// TIA Portal V20 program export: 0 tag tables, 0 data types, 60 data blocks, 132 code blocks (in call order from the OBs), 4 instance data blocks

DATA_BLOCK "DB198_eventos_generados_routing_JDT1"   // DB198
{ S7_Optimized_Access := 'FALSE' }
// stored: AutoNumber false
   VAR
      evento : Array[0..100] of String;
   END_VAR
BEGIN
END_DATA_BLOCK

DATA_BLOCK "DB202_RegEtiquetas_1001_2000"   // DB202
{ S7_Optimized_Access := 'FALSE' }
AUTHOR : ROUTER
NAME : 20130623
VERSION : 3.1
// stored: AutoNumber false
   VAR
      Reg_Etiqueta { S7_SetPoint := 'True'} : Array[1.."ROUT_Cantidad_Etiquetas_DB"] of "ROUT_Reg_Etiqueta";
   END_VAR
BEGIN
END_DATA_BLOCK

DATA_BLOCK "DB210_DB_Eventos_Router"   // DB210
{ S7_Optimized_Access := 'FALSE' }
// stored: AutoNumber false
   VAR
      EVENTO : Array[1..2600] of Char;
   END_VAR
BEGIN
END_DATA_BLOCK

DATA_BLOCK "DB211_Lecturas_Scanner"   // DB211
{ S7_Optimized_Access := 'FALSE' }
AUTHOR : ROUTER
NAME : 20130623
VERSION : 3.1
// stored: AutoNumber false
   VAR RETAIN
      Lec_Scanner { S7_SetPoint := 'True'} : Array[0.."ROUT_Max_Scanners"] of "ROUT_Datos_Lectura_Scanner";   // Num. Escaner, Long Etiquetas leidas + 1 (Primer caracter='N' nueva etiqueta).
   END_VAR
BEGIN
END_DATA_BLOCK

DATA_BLOCK "DB212_Cola_Activa"   // DB212
{ S7_Optimized_Access := 'FALSE' }
AUTHOR : ROUTER
NAME : 20130623
VERSION : 3.1
// stored: AutoNumber false
   VAR
      Cola : Array[0..9999] of UInt;   // Valor de las diferentes colas
   END_VAR
BEGIN
END_DATA_BLOCK

DATA_BLOCK "DB213_FIFO_ORDENES_SCR"   // DB213
{ S7_Optimized_Access := 'FALSE' }
AUTHOR : ROUTER
NAME : 20130623
VERSION : 3.1
// stored: AutoNumber false
   VAR
      FIFO { S7_SetPoint := 'True'} : Array[0.."ROUT_Max_Scanners"] of "ROUT_Orden_Fifo_Scanner";   // 0 a 50 scanners y 1 ordenes posibles en la FIFO
   END_VAR
BEGIN
END_DATA_BLOCK

DATA_BLOCK "DB214_CNT_Mens_SCR"   // DB214
{ S7_Optimized_Access := 'FALSE' }
AUTHOR : ROUTER
NAME : 20130623
VERSION : 3.1
// stored: AutoNumber false
   VAR RETAIN
      RedScanners : Array[1..5] of Struct
         CNT_NODO_PROF_SCR : Array[0..254] of Byte;   // No puedo acceder directamente a cargar una dirección PA de los scanners.
      END_STRUCT;
   END_VAR
BEGIN
END_DATA_BLOCK

DATA_BLOCK "DB1_SalidasExterioresDeMesa"   // DB1
{ S7_Optimized_Access := 'FALSE' }
   VAR
      Mesa { S7_SetPoint := 'True'} : Array[0.."CTE_MaxMesas"] of "UDT_SalidasExterioresDeMesa";
   END_VAR
BEGIN
END_DATA_BLOCK

DATA_BLOCK "DB220_FIFO_ORDENES_S2"   // DB220
{ S7_Optimized_Access := 'FALSE' }
AUTHOR : ROUTER
NAME : 20130623
VERSION : 3.1
// stored: AutoNumber false
   VAR
      FIFO : Array[0.."CTE_MaxMesas"] of Struct   // 0 a 50 scanners y 1 ordenes posibles en la FIFO
         Posicion { S7_SetPoint := 'True'} : Array[1..5] of "ROUT_Orden_Fifo_Scanner";
      END_STRUCT;
   END_VAR
BEGIN
END_DATA_BLOCK

DATA_BLOCK "DB230_CONTADORES"   // DB230
{ S7_Optimized_Access := 'FALSE' }
AUTHOR : ROUTER
// stored: AutoNumber false
   VAR
      Mesa : Array[0.."CTE_MaxMesas"] of Struct
         CNT_PRESENCIA : UDInt;
         CNT_AUSENCIA_ENTRADA : UDInt;
         CNT_AUSENCIA_SALIDA : UDInt;
         CNT_PARO : UDInt;
         CNT_Seg_HB_Avance : UDInt;
         CNT_Separacion_Sal : UDInt;
         CNT_Separacion_entrada : UDInt;
         CNT_CaraDelantera : UDInt;
         CNT_Reparto_E1 : UDInt;
         CNT_Reparto_E2 : UDInt;
         CNT_Reparto_E4 : UDInt;
         CNT_Detector_Fuera : UDInt;
         AUX_CNT : UDInt;
         CNT_Bloqueo_Movimiento : UDInt;
         CNT_Reposo : UDInt;
         CNT_Atasco : UDInt;
         CNT_Gap : UDInt;
         CNT_Acumulacion : UDInt;
         TMP_En_tension : UDInt;
         CNT_TopeE1S3 : UDInt;
         CNT_TopeE2S4 : UDInt;
         CNT_Transfer : UDInt;
         TMP_Decel_SM_E1S3 : UDInt;
         TMP_Decel_SM_E2S4 : UDInt;
         TMP_Decel_SM_ELEV : UDInt;
         MEM_OCUPACION : USInt;
      END_STRUCT;
   END_VAR
BEGIN
END_DATA_BLOCK

DATA_BLOCK "DB300_VelocidadesMotores"   // DB300
{ S7_Optimized_Access := 'FALSE' }
// stored: AutoNumber false
   VAR RETAIN
      TipoMotor { S7_SetPoint := 'True'} : Array[0..50] of "VelMotor";
   END_VAR
BEGIN
END_DATA_BLOCK

DATA_BLOCK "DB702_JDT02RecepMensaje"   // DB702
{ S7_Optimized_Access := 'FALSE' }
AUTHOR : TRACKING
NAME : 20130301
VERSION : 3.0
// stored: AutoNumber false
   VAR
      Mensaje : Array[0..9999] of Char;
   END_VAR
BEGIN
END_DATA_BLOCK

DATA_BLOCK "DB703_JDT02EmisionMensaje"   // DB703
{ S7_Optimized_Access := 'FALSE' }
AUTHOR : TRACKING
NAME : 20130301
VERSION : 3.0
// stored: AutoNumber false
   VAR
      Mensaje : Array[0..9999] of Char;
   END_VAR
BEGIN
END_DATA_BLOCK

DATA_BLOCK "DB704_JDT02UltimoRecibido"   // DB704
{ S7_Optimized_Access := 'FALSE' }
AUTHOR : TRACKING
NAME : 20130301
VERSION : 3.0
// stored: AutoNumber false
   VAR
      Mensaje : Array[0..9999] of Char;
   END_VAR
BEGIN
END_DATA_BLOCK

DATA_BLOCK "DB707_JDT02EventosGenerados"   // DB707
{ S7_Optimized_Access := 'FALSE' }
AUTHOR : TRACKING
NAME : 20130301
VERSION : 3.0
// stored: AutoNumber false
   VAR
      Mensaje : Array[0..9999] of Char;
   END_VAR
BEGIN
END_DATA_BLOCK

DATA_BLOCK "DB708_JDT02EventosRecibidos"   // DB708
{ S7_Optimized_Access := 'FALSE' }
AUTHOR : TRACKING
NAME : 20130301
VERSION : 3.0
// stored: AutoNumber false
   VAR
      Mensaje : Array[0..9999] of Char;
   END_VAR
BEGIN
END_DATA_BLOCK

DATA_BLOCK "DB803_JDT01EmisionMensaje"   // DB803
{ S7_Optimized_Access := 'FALSE' }
AUTHOR : TRACKING
NAME : 20130301
VERSION : 3.0
// stored: AutoNumber false
   VAR
      Mensaje : Array[0..9999] of Char;
   END_VAR
BEGIN
END_DATA_BLOCK

DATA_BLOCK "DB804_JDT01UltimoRecibido"   // DB804
{ S7_Optimized_Access := 'FALSE' }
AUTHOR : TRACKING
NAME : 20130301
VERSION : 3.0
// stored: AutoNumber false
   VAR
      Mensaje : Array[0..9999] of Char;
   END_VAR
BEGIN
END_DATA_BLOCK

DATA_BLOCK "DB807_JDT01EventosRecibidos"   // DB807
{ S7_Optimized_Access := 'FALSE' }
AUTHOR : TRACKING
NAME : 20130301
VERSION : 3.0
// stored: AutoNumber false
   VAR
      Mensaje : Array[0..9999] of Char;
   END_VAR
BEGIN
END_DATA_BLOCK

DATA_BLOCK "DB808_JDT01EventosGenerados"   // DB808
{ S7_Optimized_Access := 'FALSE' }
AUTHOR : TRACKING
NAME : 20130301
VERSION : 3.0
// stored: AutoNumber false
   VAR
      Mensaje : Array[0..9999] of Char;
   END_VAR
BEGIN
END_DATA_BLOCK

DATA_BLOCK "DB813_UTs_Ruta"   // DB813
{ S7_Optimized_Access := 'FALSE' }
AUTHOR : TRACKING
NAME : 20130301
VERSION : 3.0
// stored: AutoNumber false
   VAR
      UT { S7_SetPoint := 'True'} : Array[0.."CTE_MaxUTs"] of "UDT_UTs_Ruta";   // Array de UT's - Ruta de la UT
   END_VAR
BEGIN
END_DATA_BLOCK

DATA_BLOCK "DB814_UTs_Etiqueta"   // DB814
{ S7_Optimized_Access := 'FALSE' }
AUTHOR : TRACKING
NAME : 20130301
VERSION : 3.0
// stored: AutoNumber false
   VAR
      UT { S7_SetPoint := 'True'} : Array[0.."CTE_MaxUTs"] of "UDT_UTs_Etiqueta";   // Array de UT's - Ruta de la UT
   END_VAR
BEGIN
END_DATA_BLOCK

DATA_BLOCK "DB816_UTs_TextoPantalla"   // DB816
{ S7_Optimized_Access := 'FALSE' }
AUTHOR : TRACKING
NAME : 20130301
VERSION : 3.0
// stored: AutoNumber false
   VAR
      UT { S7_SetPoint := 'True'} : Array[0.."CTE_MaxUTs"] of "UDT_UTs_TextoPantalla";   // Array de UT's - Ruta de la UT
   END_VAR
BEGIN
END_DATA_BLOCK

DATA_BLOCK "DB820_UTs_DatosQUBIQA"   // DB820
{ S7_Optimized_Access := 'FALSE' }
AUTHOR : TRACKING
NAME : 20130301
VERSION : 3.0
// stored: AutoNumber false
   VAR
      UT { S7_SetPoint := 'True'} : Array[0.."CTE_MaxUTs"] of "UDT_UTs_DatosQUBIQA";   // Array de UT's - Ruta de la UT
   END_VAR
BEGIN
END_DATA_BLOCK

DATA_BLOCK "DB842_EmisionPantalla"   // DB842
{ S7_Optimized_Access := 'FALSE' }
// stored: AutoNumber false
BEGIN
END_DATA_BLOCK

DATA_BLOCK "DB843_RecepcionPantalla"   // DB843
{ S7_Optimized_Access := 'FALSE' }
AUTHOR : TRACKING
NAME : 20130301
VERSION : 3.0
// stored: AutoNumber false
   VAR
      Mesa { S7_SetPoint := 'True'} : Array[0.."CTE_MaxMesas"] of "UDT_ProtocoloRecDispositivo";   // Variable provisional
   END_VAR
BEGIN
END_DATA_BLOCK

DATA_BLOCK "DB891_VariablesTCP"   // DB891
{ S7_Optimized_Access := 'FALSE' }
AUTHOR : TRACKING
NAME : 20130301
VERSION : 3.0
// stored: AutoNumber false
   VAR
      TCON_JdT_PLC_Req : Bool;
      TCON_JdT_PLC_Done : Bool;
      TCON_JdT_PLC_Busy : Bool;
      TCON_JdT_PLC_Error : Bool;
      TCON_JdT_PLC_Flanco : Bool;
      Bit_05 : Bool;
      Bit_06 : Bool;
      Bit_07 : Bool;
      TDISCON_JdT_PLC_Req : Bool;
      TDISCON_JdT_PLC_Done : Bool;
      TDISCON_JdT_PLC_Busy : Bool;
      TDISCON_JdT_PLC_Error : Bool;
      TDISCON_JdT_PLC_Flanco : Bool;
      Bit_15 : Bool;
      Bit_16 : Bool;
      Bit_17 : Bool;
      TSEND_JdT_PLC_Req : Bool := TRUE;
      TSEND_JdT_PLC_Done : Bool;
      TSEND_JdT_PLC_Busy : Bool;
      TSEND_JdT_PLC_Error : Bool;
      TSEND_JdT_PLC_Flanco : Bool;
      Bit_25 : Bool;
      Bit_26 : Bool;
      Bit_27 : Bool;
      TRCV_JdT_PLC_Req : Bool;
      TRCV_JdT_PLC_Done : Bool;
      TRCV_JdT_PLC_Busy : Bool;
      TRCV_JdT_PLC_Error : Bool;
      Bit_34 : Bool;
      Bit_35 : Bool;
      Bit_36 : Bool;
      Bit_37 : Bool;
      TCON_JdT_PLC_Status : Word;
      TDISCON_JdT_PLC_Status : Word;
      TSEND_JdT_PLC_Status : Word;
      TRCV_JdT_PLC_Status : Word;
      TCON_JdT_PLC_MStatus : Word;
      TDISCON_JdT_PLC_MStatus : Word;
      TSEND_JdT_PLC_MStatus : Word;
      TRCV_JdT_PLC_MStatus : Word;
      TSEND_JdT_PLC_Longitud : Int;
      TRCV_JdT_PLC_Longitud : Int;
      TCON_JdT_PLC_Req_JDT02 : Bool;
      TCON_JdT_PLC_Done_JDT02 : Bool;
      TCON_JdT_PLC_Busy_JDT02 : Bool;
      TCON_JdT_PLC_Error_JDT02 : Bool;
      TCON_JdT_PLC_Flanco_JDT02 : Bool;
      Bit_6 : Bool;
      Bit_7 : Bool;
      Bit_8 : Bool;
      TDISCON_JdT_PLC_Req_JDT02 : Bool;
      TDISCON_JdT_PLC_Done_JDT02 : Bool;
      TDISCON_JdT_PLC_Busy_JDT02 : Bool;
      TDISCON_JdT_PLC_Error_JDT02 : Bool;
      TDISCON_JdT_PLC_Flanco_JDT02 : Bool;
      Bit_18 : Bool;
      Bit_19 : Bool;
      Bit_20 : Bool;
      TSEND_JdT_PLC_Req_JDT02 : Bool := TRUE;
      TSEND_JdT_PLC_Done_JDT02 : Bool;
      TSEND_JdT_PLC_Busy_JDT02 : Bool;
      TSEND_JdT_PLC_Error_JDT02 : Bool;
      TSEND_JdT_PLC_Flanco_JDT02 : Bool;
      Bit_28 : Bool;
      Bit_29 : Bool;
      Bit_30 : Bool;
      TRCV_JdT_PLC_Req_JDT02 : Bool;
      TRCV_JdT_PLC_Done_JDT02 : Bool;
      TRCV_JdT_PLC_Busy_JDT02 : Bool;
      TRCV_JdT_PLC_Error_JDT02 : Bool;
      Bit_38 : Bool;
      Bit_39 : Bool;
      Bit_40 : Bool;
      Bit_41 : Bool;
      TCON_JdT_PLC_Status_JDT02 : Word;
      TDISCON_JdT_PLC_Status_JDT02 : Word;
      TSEND_JdT_PLC_Status_JDT02 : Word;
      TRCV_JdT_PLC_Status_JDT02 : Word;
      TCON_JdT_PLC_MStatus_JDT02 : Word;
      TDISCON_JdT_PLC_MStatus_JDT02 : Word;
      TSEND_JdT_PLC_MStatus_JDT02 : Word;
      TRCV_JdT_PLC_MStatus_JDT02 : Word;
      TSEND_JdT_PLC_Longitud_JDT02 : Int;
      TRCV_JdT_PLC_Longitud_JDT02 : Int;
   END_VAR
BEGIN
END_DATA_BLOCK

DATA_BLOCK "DB900_Estado_Mesas"   // DB900
{ S7_Optimized_Access := 'FALSE' }
AUTHOR : GENERAL
NAME : 20160413
VERSION : 3.1
// stored: AutoNumber false
   VAR RETAIN
      EstadoVI { S7_SetPoint := 'True'} : Array[0.."CTE_MaxMesas"] of "EstadosMesa";
      MoviManual { S7_SetPoint := 'True'} : Array[0.."CTE_MaxMesas"] of "MoviManualMesa";
   END_VAR
BEGIN
END_DATA_BLOCK

DATA_BLOCK "DB901_Estado_Zonas"   // DB901
{ S7_Optimized_Access := 'FALSE' }
AUTHOR : GENERAL
NAME : 20160413
VERSION : 3.1
// stored: AutoNumber false
   VAR RETAIN
      Maximo : Int := 100;   // Maximo Numero de Zonas
      Longitud : Int := 10;   // Tamaño de la Estructura de la Zona
      Offset : Int := 6;   // Offset de la Zona Numero 0
      EstadoZona { S7_SetPoint := 'True'} : Array[0.."CTE_MaxDispositivos"] of "UDT_EstadoZonaDispositivo";   // Zona de InterCambio de Datos con la Pantalla
   END_VAR
BEGIN
END_DATA_BLOCK

DATA_BLOCK "DB902_Estado_ZonaMesa"   // DB902
{ S7_Optimized_Access := 'FALSE' }
AUTHOR : GENERAL
NAME : 20130301
VERSION : 3.0
// stored: AutoNumber false
   VAR RETAIN
      EstadoMesas { S7_SetPoint := 'True'} : Array[0.."CTE_MaxMesas"] of "EstadoZona";   // Variable provisional
   END_VAR
BEGIN
END_DATA_BLOCK

DATA_BLOCK "DB903_Estado_ZonaMaquina"   // DB903
{ S7_Optimized_Access := 'FALSE' }
AUTHOR : GENERAL
NAME : 20130301
VERSION : 3.0
// stored: AutoNumber false
   VAR RETAIN
      EstadoMaquina : Array[0.."CTE_MaxMesas"] of "EstadoZona";   // Variable provisional
   END_VAR
BEGIN
END_DATA_BLOCK

DATA_BLOCK "DB906_Interlocks"   // DB906
{ S7_Optimized_Access := 'FALSE'; DB_Accessible_From_OPC_UA := 'FALSE' }
// stored: AutoNumber false, DBAccessibleFromOPCUA false
   VAR
      Interlock { S7_SetPoint := 'True'} : Array[1.."CTE_MaxMesas"] of "UDT_Interlock_generico";
      Interlock_manual { S7_SetPoint := 'True'} : Array[1.."CTE_MaxMesas"] of "UDT_Interlock_manual";
   END_VAR
BEGIN
END_DATA_BLOCK

DATA_BLOCK "DB907_TextoErrorJdT"   // DB907
{ S7_Optimized_Access := 'FALSE' }
// stored: AutoNumber false
   VAR
      Mesa : Array[0.."CTE_MaxMesas"] of Struct
         TextoErrorJdT : String[48];
      END_STRUCT;
   END_VAR
BEGIN
END_DATA_BLOCK

DATA_BLOCK "DB936_Datos_VAR_DANFOSS_PN"   // DB936
{ S7_Optimized_Access := 'FALSE' }
// stored: AutoNumber false
   VAR RETAIN
      Danfoss : Array[0..255] of Struct
         STW_Danfoss { S7_SetPoint := 'True'} : "Danfoss_STW_PN";
         Actual_Speed : Int;
         Dig_Input { S7_SetPoint := 'True'} : "Danfoss_Dig_Input_PN";
         ACC : Int;   // 50->0,5sg; 100->1sg; 500->5sg; 1000->10sg
         DCC : Int;   // 50->0,5sg; 100->1sg; 500->5sg; 1000->10sg
      END_STRUCT;
   END_VAR
BEGIN
   Danfoss[0..255].ACC := 50;
   Danfoss[0..255].DCC := 50;
END_DATA_BLOCK

DATA_BLOCK "DB941_Datos_VAR_Lenze_i550_ASi"   // DB941
{ S7_Optimized_Access := 'FALSE' }
// stored: AutoNumber false
   VAR
      Lenze_i550 { S7_SetPoint := 'True'} : Array[1..50] of "i550 Lenze_AS-i";
   END_VAR
BEGIN
END_DATA_BLOCK

DATA_BLOCK "DB1904_Datos_Config_Gateways"   // DB1904
{ S7_Optimized_Access := 'TRUE' }
// stored: AutoNumber false, MemoryReserve 100
   VAR RETAIN
      Gateway { ExternalAccessible := 'False'; ExternalVisible := 'False'; ExternalWritable := 'False'} : Array[1..16] of Struct
         Diagnosticar { S7_SetPoint := 'True'} : Bool;   // activar el diagnosticar solo si existe
         Dos_lineas { S7_SetPoint := 'True'} : Bool;
         hwld { S7_SetPoint := 'True'} : HW_INTERFACE;
         Dir_ini_diag { S7_SetPoint := 'True'} : Int;
         Dir_ini_Asi5_L1 { S7_SetPoint := 'True'} : Int;
         Dir_ini_ASi5_L2 { S7_SetPoint := 'True'} : Int;
      END_STRUCT;
   END_VAR
BEGIN
   Gateway[1].Diagnosticar := true;
   Gateway[1].Dos_lineas := true;
   Gateway[1].hwld := 276;
   Gateway[1].Dir_ini_diag := 6000;
   Gateway[1].Dir_ini_Asi5_L1 := 600;
   Gateway[1].Dir_ini_ASi5_L2 := 900;
END_DATA_BLOCK

DATA_BLOCK "DB850_DefinicionMesas"   // DB850
{ S7_Optimized_Access := 'FALSE' }
AUTHOR : TRACKING
NAME : 20130301
VERSION : 3.0
// stored: AutoNumber false
   VAR RETAIN
      Mesa { S7_SetPoint := 'True'} : Array[0.."CTE_MaxMesas"] of "UDT_DefinicionMesa";   // Numero de Mesas que hay el Cruce de cada Mesa
   END_VAR
BEGIN
END_DATA_BLOCK

DATA_BLOCK "DB856_TipoMesaPantalla"   // DB856
{ S7_Optimized_Access := 'FALSE' }
AUTHOR : PANTALLA
NAME : 20130301
VERSION : 3.0
// stored: AutoNumber false
   VAR RETAIN
      TipoMesa : Array[0.."CTE_MaxMesas"] of Struct
         Tipo { S7_SetPoint := 'True'} : "TipoMesaPantalla";   // Tipo de Mesa para configurar la pantalla
      END_STRUCT;
   END_VAR
BEGIN
END_DATA_BLOCK

DATA_BLOCK "DB912_Tipo_Scanner_Router"   // DB912
{ S7_Optimized_Access := 'FALSE' }
AUTHOR : ROUTER
NAME : 20170522
VERSION : 3.2
// El 20170522 se incluyen las modificaciones para poder recibir y tratar mensajes INIR para varios bucles.
// stored: AutoNumber false
   VAR RETAIN
      SCANNER { S7_SetPoint := 'True'} : Array[0.."ROUT_Max_Scanners"] of "ROUT_Def_Scanner";
   END_VAR
BEGIN
   SCANNER[1..8].Tipo := 1;
   SCANNER[1].Bit_Ini_Ordenes := 1;
   SCANNER[2].Bit_Ini_Ordenes := 2;
   SCANNER[3].Bit_Ini_Ordenes := 3;
   SCANNER[4].Bit_Ini_Ordenes := 4;
   SCANNER[5].Bit_Ini_Ordenes := 5;
   SCANNER[6].Bit_Ini_Ordenes := 6;
   SCANNER[7].Bit_Ini_Ordenes := 7;
   SCANNER[8].Bit_Ini_Ordenes := 8;
   SCANNER[12].Bit_Ini_Ordenes := 7;
   SCANNER[21].Bit_Ini_Ordenes := 10;
   SCANNER[22].Bit_Ini_Ordenes := 11;
   SCANNER[23].Bit_Ini_Ordenes := 12;
   SCANNER[24].Bit_Ini_Ordenes := 13;
   SCANNER[25].Bit_Ini_Ordenes := 14;
   SCANNER[26].Bit_Ini_Ordenes := 15;
   SCANNER[27].Bit_Ini_Ordenes := 16;
   SCANNER[28].Bit_Ini_Ordenes := 17;
   SCANNER[29].Bit_Ini_Ordenes := 18;
   SCANNER[30].Bit_Ini_Ordenes := 19;
   SCANNER[31].Bit_Ini_Ordenes := 20;
   SCANNER[32].Bit_Ini_Ordenes := 21;
   SCANNER[114].Bit_Ini_Ordenes := 3;
   SCANNER[115].Bit_Ini_Ordenes := 2;
   SCANNER[116].Bit_Ini_Ordenes := 1;
   SCANNER[2..8].N_Bits_Orden := 1;
   SCANNER[1].Num_Inicializacion := -1;
   SCANNER[2].Num_Inicializacion := 2;
   SCANNER[3].Num_Inicializacion := 3;
   SCANNER[4].Num_Inicializacion := 4;
   SCANNER[5].Num_Inicializacion := 5;
   SCANNER[6].Num_Inicializacion := 6;
   SCANNER[7].Num_Inicializacion := 7;
   SCANNER[8].Num_Inicializacion := 8;
END_DATA_BLOCK

DATA_BLOCK "DB913_Router_DestinoDesvio"   // DB913
{ S7_Optimized_Access := 'FALSE' }
AUTHOR : ROUTER
NAME : 20130623
VERSION : 3.0
// stored: AutoNumber false
   VAR RETAIN
      DestinoDesvios { S7_SetPoint := 'True'} : Array[0.."ROUT_Max_Destinos"] of "ROUT_Destino_Desvios";   // Relacion de los Desvios Definidos por Destino
   END_VAR
BEGIN
END_DATA_BLOCK

DATA_BLOCK "DB990_ConfigPaletizador"   // DB990
{ S7_Optimized_Access := 'TRUE' }
// stored: AutoNumber false, MemoryReserve 100
   VAR
      Paletizador { S7_SetPoint := 'True'} : Array[1..10] of "UDT_ConfigPaletizador";
   END_VAR
BEGIN
END_DATA_BLOCK

DATA_BLOCK "DB991_ConfigDesPaletizador"   // DB991
{ S7_Optimized_Access := 'TRUE' }
// stored: AutoNumber false, MemoryReserve 100
   VAR
      Paletizador { S7_SetPoint := 'True'} : Array[1..10] of "UDT_ConfigPaletizador";
   END_VAR
BEGIN
END_DATA_BLOCK

DATA_BLOCK "DB010_ScadaConfig"   // DB10
{ S7_Optimized_Access := 'FALSE' }
AUTHOR : SCADA
NAME : 20161001
VERSION : 1.0
// stored: AutoNumber false
   VAR RETAIN
      NDB_ScadaZona : Int := 13;   // Datos del DB 13 (DB PLC ==> SCADA)
      Long_ScadaZona : Int := 24;
      OffEstado_ScadaZona : Int := 0;
      OffCodigo_ScadaZona : Int := 2;
      OffEntrada_ScadaZona : Int := 6;
      OffSalida_ScadaZona : Int := 8;
      OffDatos_ScadaZona : Int := 10;
      OffEmergGrave_ScadaZona : Int := 12;
      OffEmergLeve_ScadaZona : Int := 14;
      OffErrGrave_ScadaZona : Int := 18;
      OffErrLeve_ScadaZona : Int := 20;
   END_VAR
BEGIN
END_DATA_BLOCK

DATA_BLOCK "DB012_ScadaMaquinas"   // DB12
{ S7_Optimized_Access := 'FALSE' }
AUTHOR : SCADA
NAME : 20161001
VERSION : 1.0
// stored: AutoNumber false
   VAR
      Maquina { S7_SetPoint := 'True'} : Array[0.."CTE_MaxMesas"] of "UDT_ScadaDatosMaquina";   // MAQUINA ==> SCADA
   END_VAR
BEGIN
END_DATA_BLOCK

DATA_BLOCK "DB3000_BYPASS_SAFETY"   // DB3000, F_DB
{ S7_Optimized_Access := 'TRUE' }
// stored: AutoNumber false
   VAR
      Bypass_SF_xxxx_EM : Bool;
      Bypass_SF_xxxx_EM_1 : Bool;
      Bypass_SF_xxxx_EM_2 : Bool;
      Bypass_SF_xxxx_EM_3 : Bool;
      Bypass_SF_xxxx_EM_4 : Bool;
      Bypass_SF_xxxx_EM_5 : Bool;
      Bypass_SF_xxxx_EM_6 : Bool;
      Bypass_SF_xxxx_EM_7 : Bool;
      Bypass_SF_xxxx_EM_8 : Bool;
      Bypass_SF_xxxx_EM_9 : Bool;
      Bypass_SF_xxxx_EM_10 : Bool;
      Bypass_BF_xxBARxx : Bool;
      Bypass_BF_xxBARxx_1 : Bool;
      Bypass_BF_xxBARxx_2 : Bool;
      Bypass_BF_xxBARxx_3 : Bool;
      Bypass_BF_xxBARxx_4 : Bool;
      Bypass_BF_xxBARxx_5 : Bool;
      Bypass_BF_xxBARxx_6 : Bool;
      Bypass_SP_xxxxxx : Bool;
      Bypass_SP_xxxxxx_1 : Bool;
      Bypass_SP_xxxxxx_2 : Bool;
      Bypass_SP_xxxxxx_3 : Bool;
      Bypass_SP_xxxxxx_4 : Bool;
      Bypass_SP_xxxxxx_5 : Bool;
      Bypass_SP_xxxxxx_6 : Bool;
      Bypass_SP_xxxxxx_7 : Bool;
      Bypass_SP_xxxxxx_8 : Bool;
      Bypass_SP_xxxxxx_9 : Bool;
      Bypass_SP_xxxxxx_10 : Bool;
      Bypass_SP_xxxxxx_11 : Bool;
   END_VAR
BEGIN
END_DATA_BLOCK

DATA_BLOCK "DB9_pre_procesado"   // DB9
{ S7_Optimized_Access := 'FALSE'; DB_Accessible_From_OPC_UA := 'FALSE' }
// stored: AutoNumber false, DBAccessibleFromOPCUA false
   VAR
      marca_ciclo : "FUDT_Marcas_ciclo_seguridad";
   END_VAR
BEGIN
END_DATA_BLOCK

DATA_BLOCK "DB750_PantallaNº01"   // DB750
{ S7_Optimized_Access := 'FALSE' }
AUTHOR : PANTALLA
NAME : 20160415
VERSION : 5.0
// stored: AutoNumber false
   VAR
      HMI { S7_SetPoint := 'True'} : "UDT_HMI";
   END_VAR
BEGIN
END_DATA_BLOCK

DATA_BLOCK "DB751_PantallaNº02"   // DB751
{ S7_Optimized_Access := 'FALSE' }
AUTHOR : PANTALLA
NAME : 20160415
VERSION : 5.0
// stored: AutoNumber false
   VAR
      HMI { S7_SetPoint := 'True'} : "UDT_HMI";
   END_VAR
BEGIN
END_DATA_BLOCK

DATA_BLOCK "DB753_PantallaNº04"   // DB753
{ S7_Optimized_Access := 'FALSE' }
AUTHOR : PANTALLA
NAME : 20160415
VERSION : 5.0
// stored: AutoNumber false
   VAR
      HMI { S7_SetPoint := 'True'} : "UDT_HMI";
   END_VAR
BEGIN
END_DATA_BLOCK

DATA_BLOCK "DB754_PantallaNº05"   // DB754
{ S7_Optimized_Access := 'FALSE' }
AUTHOR : PANTALLA
NAME : 20160415
VERSION : 5.0
// stored: AutoNumber false
   VAR
      HMI { S7_SetPoint := 'True'} : "UDT_HMI";
   END_VAR
BEGIN
END_DATA_BLOCK

DATA_BLOCK "DB755_PantallaNº06"   // DB755
{ S7_Optimized_Access := 'FALSE' }
AUTHOR : PANTALLA
NAME : 20160415
VERSION : 5.0
// stored: AutoNumber false
   VAR
      HMI { S7_SetPoint := 'True'} : "UDT_HMI";
   END_VAR
BEGIN
END_DATA_BLOCK

DATA_BLOCK "DB756_PantallaNº07"   // DB756
{ S7_Optimized_Access := 'FALSE' }
AUTHOR : PANTALLA
NAME : 20160415
VERSION : 5.0
// stored: AutoNumber false
   VAR
      HMI { S7_SetPoint := 'True'} : "UDT_HMI";
   END_VAR
BEGIN
END_DATA_BLOCK

DATA_BLOCK "DB757_PantallaNº08"   // DB757
{ S7_Optimized_Access := 'FALSE' }
AUTHOR : PANTALLA
NAME : 20160415
VERSION : 5.0
// stored: AutoNumber false
   VAR
      HMI { S7_SetPoint := 'True'} : "UDT_HMI";
   END_VAR
BEGIN
END_DATA_BLOCK

DATA_BLOCK "DB758_PantallaNº09"   // DB758
{ S7_Optimized_Access := 'FALSE' }
AUTHOR : PANTALLA
NAME : 20160415
VERSION : 5.0
// stored: AutoNumber false
   VAR
      HMI { S7_SetPoint := 'True'} : "UDT_HMI";
   END_VAR
BEGIN
END_DATA_BLOCK

DATA_BLOCK "DB759_PantallaNº10"   // DB759
{ S7_Optimized_Access := 'FALSE' }
AUTHOR : PANTALLA
NAME : 20160415
VERSION : 5.0
// stored: AutoNumber false
   VAR
      HMI { S7_SetPoint := 'True'} : "UDT_HMI";
   END_VAR
BEGIN
END_DATA_BLOCK

DATA_BLOCK "DB908_Sinoptico"   // DB908
{ S7_Optimized_Access := 'FALSE' }
AUTHOR : GENERAL
NAME : 20160415
VERSION : 4.0
// stored: AutoNumber false
   VAR
      Mesa : Array[0.."CTE_MaxMesas"] of Byte;   // 0:Vacia,1:Cargada,2:EnCarga,3:EnDescarga,4:Reset,5,6,7:Error
      MesaCantidadUTs : Array[0.."CTE_MaxMesas"] of Byte;   // 0:Vacia,1:Cargada,2:EnCarga,3:EnDescarga,4:Reset,5,6,7:Error
      ArmarioPotencia : Array[0..5] of Struct   // 0:Vacia,1:Cargada,2:EnCarga,3:EnDescarga,4:Reset,5,6,7:Error
         Linea { S7_SetPoint := 'True'} : Array[0..50] of "UDT_HMI_LineaPotencia";
      END_STRUCT;
      Seta : Array[0..99] of Bool;
      BarreraQ : Array[0..99] of Bool;
      Barrera_Señales { S7_SetPoint := 'True'} : Array[0..99] of "UDT_HMI_SeñalesBarreras";
      Barrera_DIAG : Array[0..99] of Word;
      Galibo_NOOK : Array[0..29] of Bool;
      Galibo_Señal { S7_SetPoint := 'True'} : Array[0..29] of "UDT_HMI_SeñalesGalibo";
      Galibo_Codigo : Array[0..29] of Word;
      Galibo_TacoHueco : Array[0..29] of Word;
      OffsetCCPIF : UInt;
   END_VAR
BEGIN
END_DATA_BLOCK

DATA_BLOCK "DB6_Recepcion"   // DB6
{ S7_Optimized_Access := 'FALSE' }
// stored: AutoNumber false
   VAR
      ByteLIbre_000 : Byte;
      FinLote_M1 : Bool;
      Especial_M1 : Bool;
      Bit_02_M1 : Bool;
      Retroceder_M1 : Bool;
      Retirar_M1 : Bool;
      Continuar_M1 : Bool;
      Entrar_M1 : Bool;
      EmiOK_M1 : Bool;
      FinLote_M2 : Bool;
      Especial_M2 : Bool;
      Bit_02_M2 : Bool;
      Retroceder_M2 : Bool;
      Retirar_M2 : Bool;
      Continuar_M2 : Bool;
      Entrar_M2 : Bool;
      EmiOK_M2 : Bool;
      FinLote_M3 : Bool;
      Especial_M3 : Bool;
      Bit_02_M3 : Bool;
      Retroceder_M3 : Bool;
      Retirar_M3 : Bool;
      Continuar_M3 : Bool;
      Entrar_M3 : Bool;
      EmiOK_M3 : Bool;
      FinLote_M4 : Bool;
      Especial_M4 : Bool;
      Bit_02_M4 : Bool;
      Retroceder_M4 : Bool;
      Retirar_M4 : Bool;
      Continuar_M4 : Bool;
      Entrar_M4 : Bool;
      EmiOK_M4 : Bool;
      FinLote_M5 : Bool;
      Especial_M5 : Bool;
      Bit_02_M5 : Bool;
      Retroceder_M5 : Bool;
      Retirar_M5 : Bool;
      Continuar_M5 : Bool;
      Entrar_M5 : Bool;
      EmiOK_M5 : Bool;
      FinLote_M6 : Bool;
      Especial_M6 : Bool;
      Bit_02_M6 : Bool;
      Retroceder_M6 : Bool;
      Retirar_M6 : Bool;
      Continuar_M6 : Bool;
      Entrar_M6 : Bool;
      EmiOK_M6 : Bool;
      FinLote_M7 : Bool;
      Especial_M7 : Bool;
      Bit_02_M7 : Bool;
      Retroceder_M7 : Bool;
      Retirar_M7 : Bool;
      Continuar_M7 : Bool;
      Entrar_M7 : Bool;
      EmiOK_M7 : Bool;
      FinLote_M8 : Bool;
      Especial_M8 : Bool;
      Bit_02_M8 : Bool;
      Retroceder_M8 : Bool;
      Retirar_M8 : Bool;
      Continuar_M8 : Bool;
      Entrar_M8 : Bool;
      EmiOK_M8 : Bool;
      FinLote_M9 : Bool;
      Especial_M9 : Bool;
      Bit_02_M9 : Bool;
      Retroceder_M9 : Bool;
      Retirar_M9 : Bool;
      Continuar_M9 : Bool;
      Entrar_M9 : Bool;
      EmiOK_M9 : Bool;
      FinLote_M10 : Bool;
      Especial_M10 : Bool;
      Bit_02_M10 : Bool;
      Retroceder_M10 : Bool;
      Retirar_M10 : Bool;
      Continuar_M10 : Bool;
      Entrar_M10 : Bool;
      EmiOK_M10 : Bool;
      FinLote_M11 : Bool;
      Especial_M11 : Bool;
      Bit_02_M11 : Bool;
      Retroceder_M11 : Bool;
      Retirar_M11 : Bool;
      Continuar_M11 : Bool;
      Entrar_M11 : Bool;
      EmiOK_M11 : Bool;
      FinLote_M12 : Bool;
      Especial_M12 : Bool;
      Bit_02_M12 : Bool;
      Retroceder_M12 : Bool;
      Retirar_M12 : Bool;
      Continuar_M12 : Bool;
      Entrar_M12 : Bool;
      EmiOK_M12 : Bool;
      FinLote_M13 : Bool;
      Especial_M13 : Bool;
      Bit_02_M13 : Bool;
      Retroceder_M13 : Bool;
      Retirar_M13 : Bool;
      Continuar_M13 : Bool;
      Entrar_M13 : Bool;
      EmiOK_M13 : Bool;
      FinLote_M14 : Bool;
      Especial_M14 : Bool;
      Bit_02_M14 : Bool;
      Retroceder_M14 : Bool;
      Retirar_M14 : Bool;
      Continuar_M14 : Bool;
      Entrar_M14 : Bool;
      EmiOK_M14 : Bool;
      FinLote_M15 : Bool;
      Especial_M15 : Bool;
      Bit_02_M15 : Bool;
      Retroceder_M15 : Bool;
      Retirar_M15 : Bool;
      Continuar_M15 : Bool;
      Entrar_M15 : Bool;
      EmiOK_M15 : Bool;
      FinLote_M16 : Bool;
      Especial_M16 : Bool;
      Bit_02_M16 : Bool;
      Retroceder_M16 : Bool;
      Retirar_M16 : Bool;
      Continuar_M16 : Bool;
      Entrar_M16 : Bool;
      EmiOK_M16 : Bool;
      FinLote_M17 : Bool;
      Especial_M17 : Bool;
      Bit_02_M17 : Bool;
      Retroceder_M17 : Bool;
      Retirar_M17 : Bool;
      Continuar_M17 : Bool;
      Entrar_M17 : Bool;
      EmiOK_M17 : Bool;
      FinLote_M18 : Bool;
      Especial_M18 : Bool;
      Bit_02_M18 : Bool;
      Retroceder_M18 : Bool;
      Retirar_M18 : Bool;
      Continuar_M18 : Bool;
      Entrar_M18 : Bool;
      EmiOK_M18 : Bool;
      FinLote_M19 : Bool;
      Especial_M19 : Bool;
      Bit_02_M19 : Bool;
      Retroceder_M19 : Bool;
      Retirar_M19 : Bool;
      Continuar_M19 : Bool;
      Entrar_M19 : Bool;
      EmiOK_M19 : Bool;
      FinLote_M20 : Bool;
      Especial_M20 : Bool;
      Bit_02_M20 : Bool;
      Retroceder_M20 : Bool;
      Retirar_M20 : Bool;
      Continuar_M20 : Bool;
      Entrar_M20 : Bool;
      EmiOK_M20 : Bool;
      FinLote_M21 : Bool;
      Especial_M21 : Bool;
      Bit_02_M21 : Bool;
      Retroceder_M21 : Bool;
      Retirar_M21 : Bool;
      Continuar_M21 : Bool;
      Entrar_M21 : Bool;
      EmiOK_M21 : Bool;
      FinLote_M22 : Bool;
      Especial_M22 : Bool;
      Bit_02_M22 : Bool;
      Retroceder_M22 : Bool;
      Retirar_M22 : Bool;
      Continuar_M22 : Bool;
      Entrar_M22 : Bool;
      EmiOK_M22 : Bool;
      FinLote_M23 : Bool;
      Especial_M23 : Bool;
      Bit_02_M23 : Bool;
      Retroceder_M23 : Bool;
      Retirar_M23 : Bool;
      Continuar_M23 : Bool;
      Entrar_M23 : Bool;
      EmiOK_M23 : Bool;
      FinLote_M24 : Bool;
      Especial_M24 : Bool;
      Bit_02_M24 : Bool;
      Retroceder_M24 : Bool;
      Retirar_M24 : Bool;
      Continuar_M24 : Bool;
      Entrar_M24 : Bool;
      EmiOK_M24 : Bool;
      FinLote_M25 : Bool;
      Especial_M25 : Bool;
      Bit_02_M25 : Bool;
      Retroceder_M25 : Bool;
      Retirar_M25 : Bool;
      Continuar_M25 : Bool;
      Entrar_M25 : Bool;
      EmiOK_M25 : Bool;
      FinLote_M26 : Bool;
      Especial_M26 : Bool;
      Bit_02_M26 : Bool;
      Retroceder_M26 : Bool;
      Retirar_M26 : Bool;
      Continuar_M26 : Bool;
      Entrar_M26 : Bool;
      EmiOK_M26 : Bool;
      FinLote_M27 : Bool;
      Especial_M27 : Bool;
      Bit_02_M27 : Bool;
      Retroceder_M27 : Bool;
      Retirar_M27 : Bool;
      Continuar_M27 : Bool;
      Entrar_M27 : Bool;
      EmiOK_M27 : Bool;
      FinLote_M28 : Bool;
      Especial_M28 : Bool;
      Bit_02_M28 : Bool;
      Retroceder_M28 : Bool;
      Retirar_M28 : Bool;
      Continuar_M28 : Bool;
      Entrar_M28 : Bool;
      EmiOK_M28 : Bool;
      FinLote_M29 : Bool;
      Especial_M29 : Bool;
      Bit_02_M29 : Bool;
      Retroceder_M29 : Bool;
      Retirar_M29 : Bool;
      Continuar_M29 : Bool;
      Entrar_M29 : Bool;
      EmiOK_M29 : Bool;
      FinLote_M30 : Bool;
      Especial_M30 : Bool;
      Bit_02_M30 : Bool;
      Retroceder_M30 : Bool;
      Retirar_M30 : Bool;
      Continuar_M30 : Bool;
      Entrar_M30 : Bool;
      EmiOK_M30 : Bool;
      FinLote_M31 : Bool;
      Especial_M31 : Bool;
      Bit_02_M31 : Bool;
      Retroceder_M31 : Bool;
      Retirar_M31 : Bool;
      Continuar_M31 : Bool;
      Entrar_M31 : Bool;
      EmiOK_M31 : Bool;
      FinLote_M32 : Bool;
      Especial_M32 : Bool;
      Bit_02_M32 : Bool;
      Retroceder_M32 : Bool;
      Retirar_M32 : Bool;
      Continuar_M32 : Bool;
      Entrar_M32 : Bool;
      EmiOK_M32 : Bool;
      FinLote_M33 : Bool;
      Especial_M33 : Bool;
      Bit_02_M33 : Bool;
      Retroceder_M33 : Bool;
      Retirar_M33 : Bool;
      Continuar_M33 : Bool;
      Entrar_M33 : Bool;
      EmiOK_M33 : Bool;
      FinLote_M34 : Bool;
      Especial_M34 : Bool;
      Bit_02_M34 : Bool;
      Retroceder_M34 : Bool;
      Retirar_M34 : Bool;
      Continuar_M34 : Bool;
      Entrar_M34 : Bool;
      EmiOK_M34 : Bool;
      FinLote_M35 : Bool;
      Especial_M35 : Bool;
      Bit_02_M35 : Bool;
      Retroceder_M35 : Bool;
      Retirar_M35 : Bool;
      Continuar_M35 : Bool;
      Entrar_M35 : Bool;
      EmiOK_M35 : Bool;
      FinLote_M36 : Bool;
      Especial_M36 : Bool;
      Bit_02_M36 : Bool;
      Retroceder_M36 : Bool;
      Retirar_M36 : Bool;
      Continuar_M36 : Bool;
      Entrar_M36 : Bool;
      EmiOK_M36 : Bool;
      FinLote_M37 : Bool;
      Especial_M37 : Bool;
      Bit_02_M37 : Bool;
      Retroceder_M37 : Bool;
      Retirar_M37 : Bool;
      Continuar_M37 : Bool;
      Entrar_M37 : Bool;
      EmiOK_M37 : Bool;
      FinLote_M38 : Bool;
      Especial_M38 : Bool;
      Bit_02_M38 : Bool;
      Retroceder_M38 : Bool;
      Retirar_M38 : Bool;
      Continuar_M38 : Bool;
      Entrar_M38 : Bool;
      EmiOK_M38 : Bool;
      FinLote_M39 : Bool;
      Especial_M39 : Bool;
      Bit_02_M39 : Bool;
      Retroceder_M39 : Bool;
      Retirar_M39 : Bool;
      Continuar_M39 : Bool;
      Entrar_M39 : Bool;
      EmiOK_M39 : Bool;
      FinLote_M40 : Bool;
      Especial_M40 : Bool;
      Bit_02_M40 : Bool;
      Retroceder_M40 : Bool;
      Retirar_M40 : Bool;
      Continuar_M40 : Bool;
      Entrar_M40 : Bool;
      EmiOK_M40 : Bool;
      FinLote_M41 : Bool;
      Especial_M41 : Bool;
      Bit_02_M41 : Bool;
      Retroceder_M41 : Bool;
      Retirar_M41 : Bool;
      Continuar_M41 : Bool;
      Entrar_M41 : Bool;
      EmiOK_M41 : Bool;
      FinLote_M42 : Bool;
      Especial_M42 : Bool;
      Bit_02_M42 : Bool;
      Retroceder_M42 : Bool;
      Retirar_M42 : Bool;
      Continuar_M42 : Bool;
      Entrar_M42 : Bool;
      EmiOK_M42 : Bool;
      FinLote_M43 : Bool;
      Especial_M43 : Bool;
      Bit_02_M43 : Bool;
      Retroceder_M43 : Bool;
      Retirar_M43 : Bool;
      Continuar_M43 : Bool;
      Entrar_M43 : Bool;
      EmiOK_M43 : Bool;
      FinLote_M44 : Bool;
      Especial_M44 : Bool;
      Bit_02_M44 : Bool;
      Retroceder_M44 : Bool;
      Retirar_M44 : Bool;
      Continuar_M44 : Bool;
      Entrar_M44 : Bool;
      EmiOK_M44 : Bool;
      FinLote_M45 : Bool;
      Especial_M45 : Bool;
      Bit_02_M45 : Bool;
      Retroceder_M45 : Bool;
      Retirar_M45 : Bool;
      Continuar_M45 : Bool;
      Entrar_M45 : Bool;
      EmiOK_M45 : Bool;
      FinLote_M46 : Bool;
      Especial_M46 : Bool;
      Bit_02_M46 : Bool;
      Retroceder_M46 : Bool;
      Retirar_M46 : Bool;
      Continuar_M46 : Bool;
      Entrar_M46 : Bool;
      EmiOK_M46 : Bool;
      FinLote_M47 : Bool;
      Especial_M47 : Bool;
      Bit_02_M47 : Bool;
      Retroceder_M47 : Bool;
      Retirar_M47 : Bool;
      Continuar_M47 : Bool;
      Entrar_M47 : Bool;
      EmiOK_M47 : Bool;
      FinLote_M48 : Bool;
      Especial_M48 : Bool;
      Bit_02_M48 : Bool;
      Retroceder_M48 : Bool;
      Retirar_M48 : Bool;
      Continuar_M48 : Bool;
      Entrar_M48 : Bool;
      EmiOK_M48 : Bool;
      FinLote_M49 : Bool;
      Especial_M49 : Bool;
      Bit_02_M49 : Bool;
      Retroceder_M49 : Bool;
      Retirar_M49 : Bool;
      Continuar_M49 : Bool;
      Entrar_M49 : Bool;
      EmiOK_M49 : Bool;
      FinLote_M50 : Bool;
      Especial_M50 : Bool;
      Bit_02_M50 : Bool;
      Retroceder_M50 : Bool;
      Retirar_M50 : Bool;
      Continuar_M50 : Bool;
      Entrar_M50 : Bool;
      EmiOK_M50 : Bool;
      FinLote_M51 : Bool;
      Especial_M51 : Bool;
      Bit_02_M51 : Bool;
      Retroceder_M51 : Bool;
      Retirar_M51 : Bool;
      Continuar_M51 : Bool;
      Entrar_M51 : Bool;
      EmiOK_M51 : Bool;
      FinLote_M52 : Bool;
      Especial_M52 : Bool;
      Bit_02_M52 : Bool;
      Retroceder_M52 : Bool;
      Retirar_M52 : Bool;
      Continuar_M52 : Bool;
      Entrar_M52 : Bool;
      EmiOK_M52 : Bool;
      FinLote_M53 : Bool;
      Especial_M53 : Bool;
      Bit_02_M53 : Bool;
      Retroceder_M53 : Bool;
      Retirar_M53 : Bool;
      Continuar_M53 : Bool;
      Entrar_M53 : Bool;
      EmiOK_M53 : Bool;
      FinLote_M54 : Bool;
      Especial_M54 : Bool;
      Bit_02_M54 : Bool;
      Retroceder_M54 : Bool;
      Retirar_M54 : Bool;
      Continuar_M54 : Bool;
      Entrar_M54 : Bool;
      EmiOK_M54 : Bool;
      FinLote_M55 : Bool;
      Especial_M55 : Bool;
      Bit_02_M55 : Bool;
      Retroceder_M55 : Bool;
      Retirar_M55 : Bool;
      Continuar_M55 : Bool;
      Entrar_M55 : Bool;
      EmiOK_M55 : Bool;
      FinLote_M56 : Bool;
      Especial_M56 : Bool;
      Bit_02_M56 : Bool;
      Retroceder_M56 : Bool;
      Retirar_M56 : Bool;
      Continuar_M56 : Bool;
      Entrar_M56 : Bool;
      EmiOK_M56 : Bool;
      FinLote_M57 : Bool;
      Especial_M57 : Bool;
      Bit_02_M57 : Bool;
      Retroceder_M57 : Bool;
      Retirar_M57 : Bool;
      Continuar_M57 : Bool;
      Entrar_M57 : Bool;
      EmiOK_M57 : Bool;
      FinLote_M58 : Bool;
      Especial_M58 : Bool;
      Bit_02_M58 : Bool;
      Retroceder_M58 : Bool;
      Retirar_M58 : Bool;
      Continuar_M58 : Bool;
      Entrar_M58 : Bool;
      EmiOK_M58 : Bool;
      FinLote_M59 : Bool;
      Especial_M59 : Bool;
      Bit_02_M59 : Bool;
      Retroceder_M59 : Bool;
      Retirar_M59 : Bool;
      Continuar_M59 : Bool;
      Entrar_M59 : Bool;
      EmiOK_M59 : Bool;
      FinLote_M60 : Bool;
      Especial_M60 : Bool;
      Bit_02_M60 : Bool;
      Retroceder_M60 : Bool;
      Retirar_M60 : Bool;
      Continuar_M60 : Bool;
      Entrar_M60 : Bool;
      EmiOK_M60 : Bool;
      FinLote_M61 : Bool;
      Especial_M61 : Bool;
      Bit_02_M61 : Bool;
      Retroceder_M61 : Bool;
      Retirar_M61 : Bool;
      Continuar_M61 : Bool;
      Entrar_M61 : Bool;
      EmiOK_M61 : Bool;
      FinLote_M62 : Bool;
      Especial_M62 : Bool;
      Bit_02_M62 : Bool;
      Retroceder_M62 : Bool;
      Retirar_M62 : Bool;
      Continuar_M62 : Bool;
      Entrar_M62 : Bool;
      EmiOK_M62 : Bool;
      FinLote_M63 : Bool;
      Especial_M63 : Bool;
      Bit_02_M63 : Bool;
      Retroceder_M63 : Bool;
      Retirar_M63 : Bool;
      Continuar_M63 : Bool;
      Entrar_M63 : Bool;
      EmiOK_M63 : Bool;
      FinLote_M64 : Bool;
      Especial_M64 : Bool;
      Bit_02_M64 : Bool;
      Retroceder_M64 : Bool;
      Retirar_M64 : Bool;
      Continuar_M64 : Bool;
      Entrar_M64 : Bool;
      EmiOK_M64 : Bool;
      FinLote_M65 : Bool;
      Especial_M65 : Bool;
      Bit_02_M65 : Bool;
      Retroceder_M65 : Bool;
      Retirar_M65 : Bool;
      Continuar_M65 : Bool;
      Entrar_M65 : Bool;
      EmiOK_M65 : Bool;
      FinLote_M66 : Bool;
      Especial_M66 : Bool;
      Bit_02_M66 : Bool;
      Retroceder_M66 : Bool;
      Retirar_M66 : Bool;
      Continuar_M66 : Bool;
      Entrar_M66 : Bool;
      EmiOK_M66 : Bool;
      FinLote_M67 : Bool;
      Especial_M67 : Bool;
      Bit_02_M67 : Bool;
      Retroceder_M67 : Bool;
      Retirar_M67 : Bool;
      Continuar_M67 : Bool;
      Entrar_M67 : Bool;
      EmiOK_M67 : Bool;
      FinLote_M68 : Bool;
      Especial_M68 : Bool;
      Bit_02_M68 : Bool;
      Retroceder_M68 : Bool;
      Retirar_M68 : Bool;
      Continuar_M68 : Bool;
      Entrar_M68 : Bool;
      EmiOK_M68 : Bool;
      FinLote_M69 : Bool;
      Especial_M69 : Bool;
      Bit_02_M69 : Bool;
      Retroceder_M69 : Bool;
      Retirar_M69 : Bool;
      Continuar_M69 : Bool;
      Entrar_M69 : Bool;
      EmiOK_M69 : Bool;
      FinLote_M70 : Bool;
      Especial_M70 : Bool;
      Bit_02_M70 : Bool;
      Retroceder_M70 : Bool;
      Retirar_M70 : Bool;
      Continuar_M70 : Bool;
      Entrar_M70 : Bool;
      EmiOK_M70 : Bool;
      FinLote_M71 : Bool;
      Especial_M71 : Bool;
      Bit_02_M71 : Bool;
      Retroceder_M71 : Bool;
      Retirar_M71 : Bool;
      Continuar_M71 : Bool;
      Entrar_M71 : Bool;
      EmiOK_M71 : Bool;
      FinLote_M72 : Bool;
      Especial_M72 : Bool;
      Bit_02_M72 : Bool;
      Retroceder_M72 : Bool;
      Retirar_M72 : Bool;
      Continuar_M72 : Bool;
      Entrar_M72 : Bool;
      EmiOK_M72 : Bool;
      FinLote_M73 : Bool;
      Especial_M73 : Bool;
      Bit_02_M73 : Bool;
      Retroceder_M73 : Bool;
      Retirar_M73 : Bool;
      Continuar_M73 : Bool;
      Entrar_M73 : Bool;
      EmiOK_M73 : Bool;
      FinLote_M74 : Bool;
      Especial_M74 : Bool;
      Bit_02_M74 : Bool;
      Retroceder_M74 : Bool;
      Retirar_M74 : Bool;
      Continuar_M74 : Bool;
      Entrar_M74 : Bool;
      EmiOK_M74 : Bool;
      FinLote_M75 : Bool;
      Especial_M75 : Bool;
      Bit_02_M75 : Bool;
      Retroceder_M75 : Bool;
      Retirar_M75 : Bool;
      Continuar_M75 : Bool;
      Entrar_M75 : Bool;
      EmiOK_M75 : Bool;
      FinLote_M76 : Bool;
      Especial_M76 : Bool;
      Bit_02_M76 : Bool;
      Retroceder_M76 : Bool;
      Retirar_M76 : Bool;
      Continuar_M76 : Bool;
      Entrar_M76 : Bool;
      EmiOK_M76 : Bool;
      FinLote_M77 : Bool;
      Especial_M77 : Bool;
      Bit_02_M77 : Bool;
      Retroceder_M77 : Bool;
      Retirar_M77 : Bool;
      Continuar_M77 : Bool;
      Entrar_M77 : Bool;
      EmiOK_M77 : Bool;
      FinLote_M78 : Bool;
      Especial_M78 : Bool;
      Bit_02_M78 : Bool;
      Retroceder_M78 : Bool;
      Retirar_M78 : Bool;
      Continuar_M78 : Bool;
      Entrar_M78 : Bool;
      EmiOK_M78 : Bool;
      FinLote_M79 : Bool;
      Especial_M79 : Bool;
      Bit_02_M79 : Bool;
      Retroceder_M79 : Bool;
      Retirar_M79 : Bool;
      Continuar_M79 : Bool;
      Entrar_M79 : Bool;
      EmiOK_M79 : Bool;
      FinLote_M80 : Bool;
      Especial_M80 : Bool;
      Bit_02_M80 : Bool;
      Retroceder_M80 : Bool;
      Retirar_M80 : Bool;
      Continuar_M80 : Bool;
      Entrar_M80 : Bool;
      EmiOK_M80 : Bool;
      FinLote_M81 : Bool;
      Especial_M81 : Bool;
      Bit_02_M81 : Bool;
      Retroceder_M81 : Bool;
      Retirar_M81 : Bool;
      Continuar_M81 : Bool;
      Entrar_M81 : Bool;
      EmiOK_M81 : Bool;
      FinLote_M82 : Bool;
      Especial_M82 : Bool;
      Bit_02_M82 : Bool;
      Retroceder_M82 : Bool;
      Retirar_M82 : Bool;
      Continuar_M82 : Bool;
      Entrar_M82 : Bool;
      EmiOK_M82 : Bool;
      FinLote_M83 : Bool;
      Especial_M83 : Bool;
      Bit_02_M83 : Bool;
      Retroceder_M83 : Bool;
      Retirar_M83 : Bool;
      Continuar_M83 : Bool;
      Entrar_M83 : Bool;
      EmiOK_M83 : Bool;
      FinLote_M84 : Bool;
      Especial_M84 : Bool;
      Bit_02_M84 : Bool;
      Retroceder_M84 : Bool;
      Retirar_M84 : Bool;
      Continuar_M84 : Bool;
      Entrar_M84 : Bool;
      EmiOK_M84 : Bool;
      FinLote_M85 : Bool;
      Especial_M85 : Bool;
      Bit_02_M85 : Bool;
      Retroceder_M85 : Bool;
      Retirar_M85 : Bool;
      Continuar_M85 : Bool;
      Entrar_M85 : Bool;
      EmiOK_M85 : Bool;
      FinLote_M86 : Bool;
      Especial_M86 : Bool;
      Bit_02_M86 : Bool;
      Retroceder_M86 : Bool;
      Retirar_M86 : Bool;
      Continuar_M86 : Bool;
      Entrar_M86 : Bool;
      EmiOK_M86 : Bool;
      FinLote_M87 : Bool;
      Especial_M87 : Bool;
      Bit_02_M87 : Bool;
      Retroceder_M87 : Bool;
      Retirar_M87 : Bool;
      Continuar_M87 : Bool;
      Entrar_M87 : Bool;
      EmiOK_M87 : Bool;
      FinLote_M88 : Bool;
      Especial_M88 : Bool;
      Bit_02_M88 : Bool;
      Retroceder_M88 : Bool;
      Retirar_M88 : Bool;
      Continuar_M88 : Bool;
      Entrar_M88 : Bool;
      EmiOK_M88 : Bool;
      FinLote_M89 : Bool;
      Especial_M89 : Bool;
      Bit_02_M89 : Bool;
      Retroceder_M89 : Bool;
      Retirar_M89 : Bool;
      Continuar_M89 : Bool;
      Entrar_M89 : Bool;
      EmiOK_M89 : Bool;
      FinLote_M90 : Bool;
      Especial_M90 : Bool;
      Bit_02_M90 : Bool;
      Retroceder_M90 : Bool;
      Retirar_M90 : Bool;
      Continuar_M90 : Bool;
      Entrar_M90 : Bool;
      EmiOK_M90 : Bool;
      FinLote_M91 : Bool;
      Especial_M91 : Bool;
      Bit_02_M91 : Bool;
      Retroceder_M91 : Bool;
      Retirar_M91 : Bool;
      Continuar_M91 : Bool;
      Entrar_M91 : Bool;
      EmiOK_M91 : Bool;
      FinLote_M92 : Bool;
      Especial_M92 : Bool;
      Bit_02_M92 : Bool;
      Retroceder_M92 : Bool;
      Retirar_M92 : Bool;
      Continuar_M92 : Bool;
      Entrar_M92 : Bool;
      EmiOK_M92 : Bool;
      FinLote_M93 : Bool;
      Especial_M93 : Bool;
      Bit_02_M93 : Bool;
      Retroceder_M93 : Bool;
      Retirar_M93 : Bool;
      Continuar_M93 : Bool;
      Entrar_M93 : Bool;
      EmiOK_M93 : Bool;
      FinLote_M94 : Bool;
      Especial_M94 : Bool;
      Bit_02_M94 : Bool;
      Retroceder_M94 : Bool;
      Retirar_M94 : Bool;
      Continuar_M94 : Bool;
      Entrar_M94 : Bool;
      EmiOK_M94 : Bool;
      FinLote_M95 : Bool;
      Especial_M95 : Bool;
      Bit_02_M95 : Bool;
      Retroceder_M95 : Bool;
      Retirar_M95 : Bool;
      Continuar_M95 : Bool;
      Entrar_M95 : Bool;
      EmiOK_M95 : Bool;
      FinLote_M96 : Bool;
      Especial_M96 : Bool;
      Bit_02_M96 : Bool;
      Retroceder_M96 : Bool;
      Retirar_M96 : Bool;
      Continuar_M96 : Bool;
      Entrar_M96 : Bool;
      EmiOK_M96 : Bool;
      FinLote_M97 : Bool;
      Especial_M97 : Bool;
      Bit_02_M97 : Bool;
      Retroceder_M97 : Bool;
      Retirar_M97 : Bool;
      Continuar_M97 : Bool;
      Entrar_M97 : Bool;
      EmiOK_M97 : Bool;
      FinLote_M98 : Bool;
      Especial_M98 : Bool;
      Bit_02_M98 : Bool;
      Retroceder_M98 : Bool;
      Retirar_M98 : Bool;
      Continuar_M98 : Bool;
      Entrar_M98 : Bool;
      EmiOK_M98 : Bool;
      FinLote_M99 : Bool;
      Especial_M99 : Bool;
      Bit_02_M99 : Bool;
      Retroceder_M99 : Bool;
      Retirar_M99 : Bool;
      Continuar_M99 : Bool;
      Entrar_M99 : Bool;
      EmiOK_M99 : Bool;
      FinLote_M100 : Bool;
      Especial_M100 : Bool;
      Bit_02_M100 : Bool;
      Retroceder_M100 : Bool;
      Retirar_M100 : Bool;
      Continuar_M100 : Bool;
      Entrar_M100 : Bool;
      EmiOK_M100 : Bool;
      FinLote_M101 : Bool;
      Especial_M101 : Bool;
      Bit_02_M101 : Bool;
      Retroceder_M101 : Bool;
      Retirar_M101 : Bool;
      Continuar_M101 : Bool;
      Entrar_M101 : Bool;
      EmiOK_M101 : Bool;
      FinLote_M102 : Bool;
      Especial_M102 : Bool;
      Bit_02_M102 : Bool;
      Retroceder_M102 : Bool;
      Retirar_M102 : Bool;
      Continuar_M102 : Bool;
      Entrar_M102 : Bool;
      EmiOK_M102 : Bool;
      FinLote_M103 : Bool;
      Especial_M103 : Bool;
      Bit_02_M103 : Bool;
      Retroceder_M103 : Bool;
      Retirar_M103 : Bool;
      Continuar_M103 : Bool;
      Entrar_M103 : Bool;
      EmiOK_M103 : Bool;
      FinLote_M104 : Bool;
      Especial_M104 : Bool;
      Bit_02_M104 : Bool;
      Retroceder_M104 : Bool;
      Retirar_M104 : Bool;
      Continuar_M104 : Bool;
      Entrar_M104 : Bool;
      EmiOK_M104 : Bool;
      FinLote_M105 : Bool;
      Especial_M105 : Bool;
      Bit_02_M105 : Bool;
      Retroceder_M105 : Bool;
      Retirar_M105 : Bool;
      Continuar_M105 : Bool;
      Entrar_M105 : Bool;
      EmiOK_M105 : Bool;
      FinLote_M106 : Bool;
      Especial_M106 : Bool;
      Bit_02_M106 : Bool;
      Retroceder_M106 : Bool;
      Retirar_M106 : Bool;
      Continuar_M106 : Bool;
      Entrar_M106 : Bool;
      EmiOK_M106 : Bool;
      FinLote_M107 : Bool;
      Especial_M107 : Bool;
      Bit_02_M107 : Bool;
      Retroceder_M107 : Bool;
      Retirar_M107 : Bool;
      Continuar_M107 : Bool;
      Entrar_M107 : Bool;
      EmiOK_M107 : Bool;
      FinLote_M108 : Bool;
      Especial_M108 : Bool;
      Bit_02_M108 : Bool;
      Retroceder_M108 : Bool;
      Retirar_M108 : Bool;
      Continuar_M108 : Bool;
      Entrar_M108 : Bool;
      EmiOK_M108 : Bool;
      FinLote_M109 : Bool;
      Especial_M109 : Bool;
      Bit_02_M109 : Bool;
      Retroceder_M109 : Bool;
      Retirar_M109 : Bool;
      Continuar_M109 : Bool;
      Entrar_M109 : Bool;
      EmiOK_M109 : Bool;
      FinLote_M110 : Bool;
      Especial_M110 : Bool;
      Bit_02_M110 : Bool;
      Retroceder_M110 : Bool;
      Retirar_M110 : Bool;
      Continuar_M110 : Bool;
      Entrar_M110 : Bool;
      EmiOK_M110 : Bool;
      FinLote_M111 : Bool;
      Especial_M111 : Bool;
      Bit_02_M111 : Bool;
      Retroceder_M111 : Bool;
      Retirar_M111 : Bool;
      Continuar_M111 : Bool;
      Entrar_M111 : Bool;
      EmiOK_M111 : Bool;
      FinLote_M112 : Bool;
      Especial_M112 : Bool;
      Bit_02_M112 : Bool;
      Retroceder_M112 : Bool;
      Retirar_M112 : Bool;
      Continuar_M112 : Bool;
      Entrar_M112 : Bool;
      EmiOK_M112 : Bool;
      FinLote_M113 : Bool;
      Especial_M113 : Bool;
      Bit_02_M113 : Bool;
      Retroceder_M113 : Bool;
      Retirar_M113 : Bool;
      Continuar_M113 : Bool;
      Entrar_M113 : Bool;
      EmiOK_M113 : Bool;
      FinLote_M114 : Bool;
      Especial_M114 : Bool;
      Bit_02_M114 : Bool;
      Retroceder_M114 : Bool;
      Retirar_M114 : Bool;
      Continuar_M114 : Bool;
      Entrar_M114 : Bool;
      EmiOK_M114 : Bool;
      FinLote_M115 : Bool;
      Especial_M115 : Bool;
      Bit_02_M115 : Bool;
      Retroceder_M115 : Bool;
      Retirar_M115 : Bool;
      Continuar_M115 : Bool;
      Entrar_M115 : Bool;
      EmiOK_M115 : Bool;
      FinLote_M116 : Bool;
      Especial_M116 : Bool;
      Bit_02_M116 : Bool;
      Retroceder_M116 : Bool;
      Retirar_M116 : Bool;
      Continuar_M116 : Bool;
      Entrar_M116 : Bool;
      EmiOK_M116 : Bool;
      FinLote_M117 : Bool;
      Especial_M117 : Bool;
      Bit_02_M117 : Bool;
      Retroceder_M117 : Bool;
      Retirar_M117 : Bool;
      Continuar_M117 : Bool;
      Entrar_M117 : Bool;
      EmiOK_M117 : Bool;
      FinLote_M118 : Bool;
      Especial_M118 : Bool;
      Bit_02_M118 : Bool;
      Retroceder_M118 : Bool;
      Retirar_M118 : Bool;
      Continuar_M118 : Bool;
      Entrar_M118 : Bool;
      EmiOK_M118 : Bool;
      FinLote_M119 : Bool;
      Especial_M119 : Bool;
      Bit_02_M119 : Bool;
      Retroceder_M119 : Bool;
      Retirar_M119 : Bool;
      Continuar_M119 : Bool;
      Entrar_M119 : Bool;
      EmiOK_M119 : Bool;
      FinLote_M120 : Bool;
      Especial_M120 : Bool;
      Bit_02_M120 : Bool;
      Retroceder_M120 : Bool;
      Retirar_M120 : Bool;
      Continuar_M120 : Bool;
      Entrar_M120 : Bool;
      EmiOK_M120 : Bool;
      FinLote_M121 : Bool;
      Especial_M121 : Bool;
      Bit_02_M121 : Bool;
      Retroceder_M121 : Bool;
      Retirar_M121 : Bool;
      Continuar_M121 : Bool;
      Entrar_M121 : Bool;
      EmiOK_M121 : Bool;
      FinLote_M122 : Bool;
      Especial_M122 : Bool;
      Bit_02_M122 : Bool;
      Retroceder_M122 : Bool;
      Retirar_M122 : Bool;
      Continuar_M122 : Bool;
      Entrar_M122 : Bool;
      EmiOK_M122 : Bool;
      FinLote_M123 : Bool;
      Especial_M123 : Bool;
      Bit_02_M123 : Bool;
      Retroceder_M123 : Bool;
      Retirar_M123 : Bool;
      Continuar_M123 : Bool;
      Entrar_M123 : Bool;
      EmiOK_M123 : Bool;
      FinLote_M124 : Bool;
      Especial_M124 : Bool;
      Bit_02_M124 : Bool;
      Retroceder_M124 : Bool;
      Retirar_M124 : Bool;
      Continuar_M124 : Bool;
      Entrar_M124 : Bool;
      EmiOK_M124 : Bool;
      FinLote_M125 : Bool;
      Especial_M125 : Bool;
      Bit_02_M125 : Bool;
      Retroceder_M125 : Bool;
      Retirar_M125 : Bool;
      Continuar_M125 : Bool;
      Entrar_M125 : Bool;
      EmiOK_M125 : Bool;
      FinLote_M126 : Bool;
      Especial_M126 : Bool;
      Bit_02_M126 : Bool;
      Retroceder_M126 : Bool;
      Retirar_M126 : Bool;
      Continuar_M126 : Bool;
      Entrar_M126 : Bool;
      EmiOK_M126 : Bool;
      FinLote_M127 : Bool;
      Especial_M127 : Bool;
      Bit_02_M127 : Bool;
      Retroceder_M127 : Bool;
      Retirar_M127 : Bool;
      Continuar_M127 : Bool;
      Entrar_M127 : Bool;
      EmiOK_M127 : Bool;
      FinLote_M128 : Bool;
      Especial_M128 : Bool;
      Bit_02_M128 : Bool;
      Retroceder_M128 : Bool;
      Retirar_M128 : Bool;
      Continuar_M128 : Bool;
      Entrar_M128 : Bool;
      EmiOK_M128 : Bool;
      FinLote_M129 : Bool;
      Especial_M129 : Bool;
      Bit_02_M129 : Bool;
      Retroceder_M129 : Bool;
      Retirar_M129 : Bool;
      Continuar_M129 : Bool;
      Entrar_M129 : Bool;
      EmiOK_M129 : Bool;
      FinLote_M130 : Bool;
      Especial_M130 : Bool;
      Bit_02_M130 : Bool;
      Retroceder_M130 : Bool;
      Retirar_M130 : Bool;
      Continuar_M130 : Bool;
      Entrar_M130 : Bool;
      EmiOK_M130 : Bool;
      FinLote_M131 : Bool;
      Especial_M131 : Bool;
      Bit_02_M131 : Bool;
      Retroceder_M131 : Bool;
      Retirar_M131 : Bool;
      Continuar_M131 : Bool;
      Entrar_M131 : Bool;
      EmiOK_M131 : Bool;
      FinLote_M132 : Bool;
      Especial_M132 : Bool;
      Bit_02_M132 : Bool;
      Retroceder_M132 : Bool;
      Retirar_M132 : Bool;
      Continuar_M132 : Bool;
      Entrar_M132 : Bool;
      EmiOK_M132 : Bool;
      FinLote_M133 : Bool;
      Especial_M133 : Bool;
      Bit_02_M133 : Bool;
      Retroceder_M133 : Bool;
      Retirar_M133 : Bool;
      Continuar_M133 : Bool;
      Entrar_M133 : Bool;
      EmiOK_M133 : Bool;
      FinLote_M134 : Bool;
      Especial_M134 : Bool;
      Bit_02_M134 : Bool;
      Retroceder_M134 : Bool;
      Retirar_M134 : Bool;
      Continuar_M134 : Bool;
      Entrar_M134 : Bool;
      EmiOK_M134 : Bool;
      FinLote_M135 : Bool;
      Especial_M135 : Bool;
      Bit_02_M135 : Bool;
      Retroceder_M135 : Bool;
      Retirar_M135 : Bool;
      Continuar_M135 : Bool;
      Entrar_M135 : Bool;
      EmiOK_M135 : Bool;
      FinLote_M136 : Bool;
      Especial_M136 : Bool;
      Bit_02_M136 : Bool;
      Retroceder_M136 : Bool;
      Retirar_M136 : Bool;
      Continuar_M136 : Bool;
      Entrar_M136 : Bool;
      EmiOK_M136 : Bool;
      FinLote_M137 : Bool;
      Especial_M137 : Bool;
      Bit_02_M137 : Bool;
      Retroceder_M137 : Bool;
      Retirar_M137 : Bool;
      Continuar_M137 : Bool;
      Entrar_M137 : Bool;
      EmiOK_M137 : Bool;
      FinLote_M138 : Bool;
      Especial_M138 : Bool;
      Bit_02_M138 : Bool;
      Retroceder_M138 : Bool;
      Retirar_M138 : Bool;
      Continuar_M138 : Bool;
      Entrar_M138 : Bool;
      EmiOK_M138 : Bool;
      FinLote_M139 : Bool;
      Especial_M139 : Bool;
      Bit_02_M139 : Bool;
      Retroceder_M139 : Bool;
      Retirar_M139 : Bool;
      Continuar_M139 : Bool;
      Entrar_M139 : Bool;
      EmiOK_M139 : Bool;
      FinLote_M140 : Bool;
      Especial_M140 : Bool;
      Bit_02_M140 : Bool;
      Retroceder_M140 : Bool;
      Retirar_M140 : Bool;
      Continuar_M140 : Bool;
      Entrar_M140 : Bool;
      EmiOK_M140 : Bool;
      FinLote_M141 : Bool;
      Especial_M141 : Bool;
      Bit_02_M141 : Bool;
      Retroceder_M141 : Bool;
      Retirar_M141 : Bool;
      Continuar_M141 : Bool;
      Entrar_M141 : Bool;
      EmiOK_M141 : Bool;
      FinLote_M142 : Bool;
      Especial_M142 : Bool;
      Bit_02_M142 : Bool;
      Retroceder_M142 : Bool;
      Retirar_M142 : Bool;
      Continuar_M142 : Bool;
      Entrar_M142 : Bool;
      EmiOK_M142 : Bool;
      FinLote_M143 : Bool;
      Especial_M143 : Bool;
      Bit_02_M143 : Bool;
      Retroceder_M143 : Bool;
      Retirar_M143 : Bool;
      Continuar_M143 : Bool;
      Entrar_M143 : Bool;
      EmiOK_M143 : Bool;
      FinLote_M144 : Bool;
      Especial_M144 : Bool;
      Bit_02_M144 : Bool;
      Retroceder_M144 : Bool;
      Retirar_M144 : Bool;
      Continuar_M144 : Bool;
      Entrar_M144 : Bool;
      EmiOK_M144 : Bool;
      FinLote_M145 : Bool;
      Especial_M145 : Bool;
      Bit_02_M145 : Bool;
      Retroceder_M145 : Bool;
      Retirar_M145 : Bool;
      Continuar_M145 : Bool;
      Entrar_M145 : Bool;
      EmiOK_M145 : Bool;
      FinLote_M146 : Bool;
      Especial_M146 : Bool;
      Bit_02_M146 : Bool;
      Retroceder_M146 : Bool;
      Retirar_M146 : Bool;
      Continuar_M146 : Bool;
      Entrar_M146 : Bool;
      EmiOK_M146 : Bool;
      FinLote_M147 : Bool;
      Especial_M147 : Bool;
      Bit_02_M147 : Bool;
      Retroceder_M147 : Bool;
      Retirar_M147 : Bool;
      Continuar_M147 : Bool;
      Entrar_M147 : Bool;
      EmiOK_M147 : Bool;
      FinLote_M148 : Bool;
      Especial_M148 : Bool;
      Bit_02_M148 : Bool;
      Retroceder_M148 : Bool;
      Retirar_M148 : Bool;
      Continuar_M148 : Bool;
      Entrar_M148 : Bool;
      EmiOK_M148 : Bool;
      FinLote_M149 : Bool;
      Especial_M149 : Bool;
      Bit_02_M149 : Bool;
      Retroceder_M149 : Bool;
      Retirar_M149 : Bool;
      Continuar_M149 : Bool;
      Entrar_M149 : Bool;
      EmiOK_M149 : Bool;
      FinLote_M150 : Bool;
      Especial_M150 : Bool;
      Bit_02_M150 : Bool;
      Retroceder_M150 : Bool;
      Retirar_M150 : Bool;
      Continuar_M150 : Bool;
      Entrar_M150 : Bool;
      EmiOK_M150 : Bool;
      FinLote_M151 : Bool;
      Especial_M151 : Bool;
      Bit_02_M151 : Bool;
      Retroceder_M151 : Bool;
      Retirar_M151 : Bool;
      Continuar_M151 : Bool;
      Entrar_M151 : Bool;
      EmiOK_M151 : Bool;
      FinLote_M152 : Bool;
      Especial_M152 : Bool;
      Bit_02_M152 : Bool;
      Retroceder_M152 : Bool;
      Retirar_M152 : Bool;
      Continuar_M152 : Bool;
      Entrar_M152 : Bool;
      EmiOK_M152 : Bool;
      FinLote_M153 : Bool;
      Especial_M153 : Bool;
      Bit_02_M153 : Bool;
      Retroceder_M153 : Bool;
      Retirar_M153 : Bool;
      Continuar_M153 : Bool;
      Entrar_M153 : Bool;
      EmiOK_M153 : Bool;
      FinLote_M154 : Bool;
      Especial_M154 : Bool;
      Bit_02_M154 : Bool;
      Retroceder_M154 : Bool;
      Retirar_M154 : Bool;
      Continuar_M154 : Bool;
      Entrar_M154 : Bool;
      EmiOK_M154 : Bool;
      FinLote_M155 : Bool;
      Especial_M155 : Bool;
      Bit_02_M155 : Bool;
      Retroceder_M155 : Bool;
      Retirar_M155 : Bool;
      Continuar_M155 : Bool;
      Entrar_M155 : Bool;
      EmiOK_M155 : Bool;
      FinLote_M156 : Bool;
      Especial_M156 : Bool;
      Bit_02_M156 : Bool;
      Retroceder_M156 : Bool;
      Retirar_M156 : Bool;
      Continuar_M156 : Bool;
      Entrar_M156 : Bool;
      EmiOK_M156 : Bool;
      FinLote_M157 : Bool;
      Especial_M157 : Bool;
      Bit_02_M157 : Bool;
      Retroceder_M157 : Bool;
      Retirar_M157 : Bool;
      Continuar_M157 : Bool;
      Entrar_M157 : Bool;
      EmiOK_M157 : Bool;
      FinLote_M158 : Bool;
      Especial_M158 : Bool;
      Bit_02_M158 : Bool;
      Retroceder_M158 : Bool;
      Retirar_M158 : Bool;
      Continuar_M158 : Bool;
      Entrar_M158 : Bool;
      EmiOK_M158 : Bool;
      FinLote_M159 : Bool;
      Especial_M159 : Bool;
      Bit_02_M159 : Bool;
      Retroceder_M159 : Bool;
      Retirar_M159 : Bool;
      Continuar_M159 : Bool;
      Entrar_M159 : Bool;
      EmiOK_M159 : Bool;
      FinLote_M160 : Bool;
      Especial_M160 : Bool;
      Bit_02_M160 : Bool;
      Retroceder_M160 : Bool;
      Retirar_M160 : Bool;
      Continuar_M160 : Bool;
      Entrar_M160 : Bool;
      EmiOK_M160 : Bool;
      FinLote_M161 : Bool;
      Especial_M161 : Bool;
      Bit_02_M161 : Bool;
      Retroceder_M161 : Bool;
      Retirar_M161 : Bool;
      Continuar_M161 : Bool;
      Entrar_M161 : Bool;
      EmiOK_M161 : Bool;
      FinLote_M162 : Bool;
      Especial_M162 : Bool;
      Bit_02_M162 : Bool;
      Retroceder_M162 : Bool;
      Retirar_M162 : Bool;
      Continuar_M162 : Bool;
      Entrar_M162 : Bool;
      EmiOK_M162 : Bool;
      FinLote_M163 : Bool;
      Especial_M163 : Bool;
      Bit_02_M163 : Bool;
      Retroceder_M163 : Bool;
      Retirar_M163 : Bool;
      Continuar_M163 : Bool;
      Entrar_M163 : Bool;
      EmiOK_M163 : Bool;
      FinLote_M164 : Bool;
      Especial_M164 : Bool;
      Bit_02_M164 : Bool;
      Retroceder_M164 : Bool;
      Retirar_M164 : Bool;
      Continuar_M164 : Bool;
      Entrar_M164 : Bool;
      EmiOK_M164 : Bool;
      FinLote_M165 : Bool;
      Especial_M165 : Bool;
      Bit_02_M165 : Bool;
      Retroceder_M165 : Bool;
      Retirar_M165 : Bool;
      Continuar_M165 : Bool;
      Entrar_M165 : Bool;
      EmiOK_M165 : Bool;
      FinLote_M166 : Bool;
      Especial_M166 : Bool;
      Bit_02_M166 : Bool;
      Retroceder_M166 : Bool;
      Retirar_M166 : Bool;
      Continuar_M166 : Bool;
      Entrar_M166 : Bool;
      EmiOK_M166 : Bool;
      FinLote_M167 : Bool;
      Especial_M167 : Bool;
      Bit_02_M167 : Bool;
      Retroceder_M167 : Bool;
      Retirar_M167 : Bool;
      Continuar_M167 : Bool;
      Entrar_M167 : Bool;
      EmiOK_M167 : Bool;
      FinLote_M168 : Bool;
      Especial_M168 : Bool;
      Bit_02_M168 : Bool;
      Retroceder_M168 : Bool;
      Retirar_M168 : Bool;
      Continuar_M168 : Bool;
      Entrar_M168 : Bool;
      EmiOK_M168 : Bool;
      FinLote_M169 : Bool;
      Especial_M169 : Bool;
      Bit_02_M169 : Bool;
      Retroceder_M169 : Bool;
      Retirar_M169 : Bool;
      Continuar_M169 : Bool;
      Entrar_M169 : Bool;
      EmiOK_M169 : Bool;
      FinLote_M170 : Bool;
      Especial_M170 : Bool;
      Bit_02_M170 : Bool;
      Retroceder_M170 : Bool;
      Retirar_M170 : Bool;
      Continuar_M170 : Bool;
      Entrar_M170 : Bool;
      EmiOK_M170 : Bool;
      FinLote_M171 : Bool;
      Especial_M171 : Bool;
      Bit_02_M171 : Bool;
      Retroceder_M171 : Bool;
      Retirar_M171 : Bool;
      Continuar_M171 : Bool;
      Entrar_M171 : Bool;
      EmiOK_M171 : Bool;
      FinLote_M172 : Bool;
      Especial_M172 : Bool;
      Bit_02_M172 : Bool;
      Retroceder_M172 : Bool;
      Retirar_M172 : Bool;
      Continuar_M172 : Bool;
      Entrar_M172 : Bool;
      EmiOK_M172 : Bool;
      FinLote_M173 : Bool;
      Especial_M173 : Bool;
      Bit_02_M173 : Bool;
      Retroceder_M173 : Bool;
      Retirar_M173 : Bool;
      Continuar_M173 : Bool;
      Entrar_M173 : Bool;
      EmiOK_M173 : Bool;
      FinLote_M174 : Bool;
      Especial_M174 : Bool;
      Bit_02_M174 : Bool;
      Retroceder_M174 : Bool;
      Retirar_M174 : Bool;
      Continuar_M174 : Bool;
      Entrar_M174 : Bool;
      EmiOK_M174 : Bool;
      FinLote_M175 : Bool;
      Especial_M175 : Bool;
      Bit_02_M175 : Bool;
      Retroceder_M175 : Bool;
      Retirar_M175 : Bool;
      Continuar_M175 : Bool;
      Entrar_M175 : Bool;
      EmiOK_M175 : Bool;
      FinLote_M176 : Bool;
      Especial_M176 : Bool;
      Bit_02_M176 : Bool;
      Retroceder_M176 : Bool;
      Retirar_M176 : Bool;
      Continuar_M176 : Bool;
      Entrar_M176 : Bool;
      EmiOK_M176 : Bool;
      FinLote_M177 : Bool;
      Especial_M177 : Bool;
      Bit_02_M177 : Bool;
      Retroceder_M177 : Bool;
      Retirar_M177 : Bool;
      Continuar_M177 : Bool;
      Entrar_M177 : Bool;
      EmiOK_M177 : Bool;
      FinLote_M178 : Bool;
      Especial_M178 : Bool;
      Bit_02_M178 : Bool;
      Retroceder_M178 : Bool;
      Retirar_M178 : Bool;
      Continuar_M178 : Bool;
      Entrar_M178 : Bool;
      EmiOK_M178 : Bool;
      FinLote_M179 : Bool;
      Especial_M179 : Bool;
      Bit_02_M179 : Bool;
      Retroceder_M179 : Bool;
      Retirar_M179 : Bool;
      Continuar_M179 : Bool;
      Entrar_M179 : Bool;
      EmiOK_M179 : Bool;
      FinLote_M180 : Bool;
      Especial_M180 : Bool;
      Bit_02_M180 : Bool;
      Retroceder_M180 : Bool;
      Retirar_M180 : Bool;
      Continuar_M180 : Bool;
      Entrar_M180 : Bool;
      EmiOK_M180 : Bool;
      FinLote_M181 : Bool;
      Especial_M181 : Bool;
      Bit_02_M181 : Bool;
      Retroceder_M181 : Bool;
      Retirar_M181 : Bool;
      Continuar_M181 : Bool;
      Entrar_M181 : Bool;
      EmiOK_M181 : Bool;
      FinLote_M182 : Bool;
      Especial_M182 : Bool;
      Bit_02_M182 : Bool;
      Retroceder_M182 : Bool;
      Retirar_M182 : Bool;
      Continuar_M182 : Bool;
      Entrar_M182 : Bool;
      EmiOK_M182 : Bool;
      FinLote_M183 : Bool;
      Especial_M183 : Bool;
      Bit_02_M183 : Bool;
      Retroceder_M183 : Bool;
      Retirar_M183 : Bool;
      Continuar_M183 : Bool;
      Entrar_M183 : Bool;
      EmiOK_M183 : Bool;
      FinLote_M184 : Bool;
      Especial_M184 : Bool;
      Bit_02_M184 : Bool;
      Retroceder_M184 : Bool;
      Retirar_M184 : Bool;
      Continuar_M184 : Bool;
      Entrar_M184 : Bool;
      EmiOK_M184 : Bool;
      FinLote_M185 : Bool;
      Especial_M185 : Bool;
      Bit_02_M185 : Bool;
      Retroceder_M185 : Bool;
      Retirar_M185 : Bool;
      Continuar_M185 : Bool;
      Entrar_M185 : Bool;
      EmiOK_M185 : Bool;
      FinLote_M186 : Bool;
      Especial_M186 : Bool;
      Bit_02_M186 : Bool;
      Retroceder_M186 : Bool;
      Retirar_M186 : Bool;
      Continuar_M186 : Bool;
      Entrar_M186 : Bool;
      EmiOK_M186 : Bool;
      FinLote_M187 : Bool;
      Especial_M187 : Bool;
      Bit_02_M187 : Bool;
      Retroceder_M187 : Bool;
      Retirar_M187 : Bool;
      Continuar_M187 : Bool;
      Entrar_M187 : Bool;
      EmiOK_M187 : Bool;
      FinLote_M188 : Bool;
      Especial_M188 : Bool;
      Bit_02_M188 : Bool;
      Retroceder_M188 : Bool;
      Retirar_M188 : Bool;
      Continuar_M188 : Bool;
      Entrar_M188 : Bool;
      EmiOK_M188 : Bool;
      FinLote_M189 : Bool;
      Especial_M189 : Bool;
      Bit_02_M189 : Bool;
      Retroceder_M189 : Bool;
      Retirar_M189 : Bool;
      Continuar_M189 : Bool;
      Entrar_M189 : Bool;
      EmiOK_M189 : Bool;
      FinLote_M190 : Bool;
      Especial_M190 : Bool;
      Bit_02_M190 : Bool;
      Retroceder_M190 : Bool;
      Retirar_M190 : Bool;
      Continuar_M190 : Bool;
      Entrar_M190 : Bool;
      EmiOK_M190 : Bool;
      FinLote_M191 : Bool;
      Especial_M191 : Bool;
      Bit_02_M191 : Bool;
      Retroceder_M191 : Bool;
      Retirar_M191 : Bool;
      Continuar_M191 : Bool;
      Entrar_M191 : Bool;
      EmiOK_M191 : Bool;
      FinLote_M192 : Bool;
      Especial_M192 : Bool;
      Bit_02_M192 : Bool;
      Retroceder_M192 : Bool;
      Retirar_M192 : Bool;
      Continuar_M192 : Bool;
      Entrar_M192 : Bool;
      EmiOK_M192 : Bool;
      FinLote_M193 : Bool;
      Especial_M193 : Bool;
      Bit_02_M193 : Bool;
      Retroceder_M193 : Bool;
      Retirar_M193 : Bool;
      Continuar_M193 : Bool;
      Entrar_M193 : Bool;
      EmiOK_M193 : Bool;
      FinLote_M194 : Bool;
      Especial_M194 : Bool;
      Bit_02_M194 : Bool;
      Retroceder_M194 : Bool;
      Retirar_M194 : Bool;
      Continuar_M194 : Bool;
      Entrar_M194 : Bool;
      EmiOK_M194 : Bool;
      FinLote_M195 : Bool;
      Especial_M195 : Bool;
      Bit_02_M195 : Bool;
      Retroceder_M195 : Bool;
      Retirar_M195 : Bool;
      Continuar_M195 : Bool;
      Entrar_M195 : Bool;
      EmiOK_M195 : Bool;
      FinLote_M196 : Bool;
      Especial_M196 : Bool;
      Bit_02_M196 : Bool;
      Retroceder_M196 : Bool;
      Retirar_M196 : Bool;
      Continuar_M196 : Bool;
      Entrar_M196 : Bool;
      EmiOK_M196 : Bool;
      FinLote_M197 : Bool;
      Especial_M197 : Bool;
      Bit_02_M197 : Bool;
      Retroceder_M197 : Bool;
      Retirar_M197 : Bool;
      Continuar_M197 : Bool;
      Entrar_M197 : Bool;
      EmiOK_M197 : Bool;
      FinLote_M198 : Bool;
      Especial_M198 : Bool;
      Bit_02_M198 : Bool;
      Retroceder_M198 : Bool;
      Retirar_M198 : Bool;
      Continuar_M198 : Bool;
      Entrar_M198 : Bool;
      EmiOK_M198 : Bool;
      FinLote_M199 : Bool;
      Especial_M199 : Bool;
      Bit_02_M199 : Bool;
      Retroceder_M199 : Bool;
      Retirar_M199 : Bool;
      Continuar_M199 : Bool;
      Entrar_M199 : Bool;
      EmiOK_M199 : Bool;
      FinLote_M200 : Bool;
      Especial_M200 : Bool;
      Bit_02_M200 : Bool;
      Retroceder_M200 : Bool;
      Retirar_M200 : Bool;
      Continuar_M200 : Bool;
      Entrar_M200 : Bool;
      EmiOK_M200 : Bool;
      FinLote_M201 : Bool;
      Especial_M201 : Bool;
      Bit_02_M201 : Bool;
      Retroceder_M201 : Bool;
      Retirar_M201 : Bool;
      Continuar_M201 : Bool;
      Entrar_M201 : Bool;
      EmiOK_M201 : Bool;
      FinLote_M202 : Bool;
      Especial_M202 : Bool;
      Bit_02_M202 : Bool;
      Retroceder_M202 : Bool;
      Retirar_M202 : Bool;
      Continuar_M202 : Bool;
      Entrar_M202 : Bool;
      EmiOK_M202 : Bool;
      FinLote_M203 : Bool;
      Especial_M203 : Bool;
      Bit_02_M203 : Bool;
      Retroceder_M203 : Bool;
      Retirar_M203 : Bool;
      Continuar_M203 : Bool;
      Entrar_M203 : Bool;
      EmiOK_M203 : Bool;
      FinLote_M204 : Bool;
      Especial_M204 : Bool;
      Bit_02_M204 : Bool;
      Retroceder_M204 : Bool;
      Retirar_M204 : Bool;
      Continuar_M204 : Bool;
      Entrar_M204 : Bool;
      EmiOK_M204 : Bool;
      FinLote_M205 : Bool;
      Especial_M205 : Bool;
      Bit_02_M205 : Bool;
      Retroceder_M205 : Bool;
      Retirar_M205 : Bool;
      Continuar_M205 : Bool;
      Entrar_M205 : Bool;
      EmiOK_M205 : Bool;
      FinLote_M206 : Bool;
      Especial_M206 : Bool;
      Bit_02_M206 : Bool;
      Retroceder_M206 : Bool;
      Retirar_M206 : Bool;
      Continuar_M206 : Bool;
      Entrar_M206 : Bool;
      EmiOK_M206 : Bool;
      FinLote_M207 : Bool;
      Especial_M207 : Bool;
      Bit_02_M207 : Bool;
      Retroceder_M207 : Bool;
      Retirar_M207 : Bool;
      Continuar_M207 : Bool;
      Entrar_M207 : Bool;
      EmiOK_M207 : Bool;
      FinLote_M208 : Bool;
      Especial_M208 : Bool;
      Bit_02_M208 : Bool;
      Retroceder_M208 : Bool;
      Retirar_M208 : Bool;
      Continuar_M208 : Bool;
      Entrar_M208 : Bool;
      EmiOK_M208 : Bool;
      FinLote_M209 : Bool;
      Especial_M209 : Bool;
      Bit_02_M209 : Bool;
      Retroceder_M209 : Bool;
      Retirar_M209 : Bool;
      Continuar_M209 : Bool;
      Entrar_M209 : Bool;
      EmiOK_M209 : Bool;
      FinLote_M210 : Bool;
      Especial_M210 : Bool;
      Bit_02_M210 : Bool;
      Retroceder_M210 : Bool;
      Retirar_M210 : Bool;
      Continuar_M210 : Bool;
      Entrar_M210 : Bool;
      EmiOK_M210 : Bool;
      FinLote_M211 : Bool;
      Especial_M211 : Bool;
      Bit_02_M211 : Bool;
      Retroceder_M211 : Bool;
      Retirar_M211 : Bool;
      Continuar_M211 : Bool;
      Entrar_M211 : Bool;
      EmiOK_M211 : Bool;
      FinLote_M212 : Bool;
      Especial_M212 : Bool;
      Bit_02_M212 : Bool;
      Retroceder_M212 : Bool;
      Retirar_M212 : Bool;
      Continuar_M212 : Bool;
      Entrar_M212 : Bool;
      EmiOK_M212 : Bool;
      FinLote_M213 : Bool;
      Especial_M213 : Bool;
      Bit_02_M213 : Bool;
      Retroceder_M213 : Bool;
      Retirar_M213 : Bool;
      Continuar_M213 : Bool;
      Entrar_M213 : Bool;
      EmiOK_M213 : Bool;
      FinLote_M214 : Bool;
      Especial_M214 : Bool;
      Bit_02_M214 : Bool;
      Retroceder_M214 : Bool;
      Retirar_M214 : Bool;
      Continuar_M214 : Bool;
      Entrar_M214 : Bool;
      EmiOK_M214 : Bool;
      FinLote_M215 : Bool;
      Especial_M215 : Bool;
      Bit_02_M215 : Bool;
      Retroceder_M215 : Bool;
      Retirar_M215 : Bool;
      Continuar_M215 : Bool;
      Entrar_M215 : Bool;
      EmiOK_M215 : Bool;
      FinLote_M216 : Bool;
      Especial_M216 : Bool;
      Bit_02_M216 : Bool;
      Retroceder_M216 : Bool;
      Retirar_M216 : Bool;
      Continuar_M216 : Bool;
      Entrar_M216 : Bool;
      EmiOK_M216 : Bool;
      FinLote_M217 : Bool;
      Especial_M217 : Bool;
      Bit_02_M217 : Bool;
      Retroceder_M217 : Bool;
      Retirar_M217 : Bool;
      Continuar_M217 : Bool;
      Entrar_M217 : Bool;
      EmiOK_M217 : Bool;
      FinLote_M218 : Bool;
      Especial_M218 : Bool;
      Bit_02_M218 : Bool;
      Retroceder_M218 : Bool;
      Retirar_M218 : Bool;
      Continuar_M218 : Bool;
      Entrar_M218 : Bool;
      EmiOK_M218 : Bool;
      FinLote_M219 : Bool;
      Especial_M219 : Bool;
      Bit_02_M219 : Bool;
      Retroceder_M219 : Bool;
      Retirar_M219 : Bool;
      Continuar_M219 : Bool;
      Entrar_M219 : Bool;
      EmiOK_M219 : Bool;
      FinLote_M220 : Bool;
      Especial_M220 : Bool;
      Bit_02_M220 : Bool;
      Retroceder_M220 : Bool;
      Retirar_M220 : Bool;
      Continuar_M220 : Bool;
      Entrar_M220 : Bool;
      EmiOK_M220 : Bool;
      FinLote_M221 : Bool;
      Especial_M221 : Bool;
      Bit_02_M221 : Bool;
      Retroceder_M221 : Bool;
      Retirar_M221 : Bool;
      Continuar_M221 : Bool;
      Entrar_M221 : Bool;
      EmiOK_M221 : Bool;
      FinLote_M222 : Bool;
      Especial_M222 : Bool;
      Bit_02_M222 : Bool;
      Retroceder_M222 : Bool;
      Retirar_M222 : Bool;
      Continuar_M222 : Bool;
      Entrar_M222 : Bool;
      EmiOK_M222 : Bool;
      FinLote_M223 : Bool;
      Especial_M223 : Bool;
      Bit_02_M223 : Bool;
      Retroceder_M223 : Bool;
      Retirar_M223 : Bool;
      Continuar_M223 : Bool;
      Entrar_M223 : Bool;
      EmiOK_M223 : Bool;
      FinLote_M224 : Bool;
      Especial_M224 : Bool;
      Bit_02_M224 : Bool;
      Retroceder_M224 : Bool;
      Retirar_M224 : Bool;
      Continuar_M224 : Bool;
      Entrar_M224 : Bool;
      EmiOK_M224 : Bool;
      FinLote_M225 : Bool;
      Especial_M225 : Bool;
      Bit_02_M225 : Bool;
      Retroceder_M225 : Bool;
      Retirar_M225 : Bool;
      Continuar_M225 : Bool;
      Entrar_M225 : Bool;
      EmiOK_M225 : Bool;
      FinLote_M226 : Bool;
      Especial_M226 : Bool;
      Bit_02_M226 : Bool;
      Retroceder_M226 : Bool;
      Retirar_M226 : Bool;
      Continuar_M226 : Bool;
      Entrar_M226 : Bool;
      EmiOK_M226 : Bool;
      FinLote_M227 : Bool;
      Especial_M227 : Bool;
      Bit_02_M227 : Bool;
      Retroceder_M227 : Bool;
      Retirar_M227 : Bool;
      Continuar_M227 : Bool;
      Entrar_M227 : Bool;
      EmiOK_M227 : Bool;
      FinLote_M228 : Bool;
      Especial_M228 : Bool;
      Bit_02_M228 : Bool;
      Retroceder_M228 : Bool;
      Retirar_M228 : Bool;
      Continuar_M228 : Bool;
      Entrar_M228 : Bool;
      EmiOK_M228 : Bool;
      FinLote_M229 : Bool;
      Especial_M229 : Bool;
      Bit_02_M229 : Bool;
      Retroceder_M229 : Bool;
      Retirar_M229 : Bool;
      Continuar_M229 : Bool;
      Entrar_M229 : Bool;
      EmiOK_M229 : Bool;
      FinLote_M230 : Bool;
      Especial_M230 : Bool;
      Bit_02_M230 : Bool;
      Retroceder_M230 : Bool;
      Retirar_M230 : Bool;
      Continuar_M230 : Bool;
      Entrar_M230 : Bool;
      EmiOK_M230 : Bool;
      FinLote_M231 : Bool;
      Especial_M231 : Bool;
      Bit_02_M231 : Bool;
      Retroceder_M231 : Bool;
      Retirar_M231 : Bool;
      Continuar_M231 : Bool;
      Entrar_M231 : Bool;
      EmiOK_M231 : Bool;
      FinLote_M232 : Bool;
      Especial_M232 : Bool;
      Bit_02_M232 : Bool;
      Retroceder_M232 : Bool;
      Retirar_M232 : Bool;
      Continuar_M232 : Bool;
      Entrar_M232 : Bool;
      EmiOK_M232 : Bool;
      FinLote_M233 : Bool;
      Especial_M233 : Bool;
      Bit_02_M233 : Bool;
      Retroceder_M233 : Bool;
      Retirar_M233 : Bool;
      Continuar_M233 : Bool;
      Entrar_M233 : Bool;
      EmiOK_M233 : Bool;
      FinLote_M234 : Bool;
      Especial_M234 : Bool;
      Bit_02_M234 : Bool;
      Retroceder_M234 : Bool;
      Retirar_M234 : Bool;
      Continuar_M234 : Bool;
      Entrar_M234 : Bool;
      EmiOK_M234 : Bool;
      FinLote_M235 : Bool;
      Especial_M235 : Bool;
      Bit_02_M235 : Bool;
      Retroceder_M235 : Bool;
      Retirar_M235 : Bool;
      Continuar_M235 : Bool;
      Entrar_M235 : Bool;
      EmiOK_M235 : Bool;
      FinLote_M236 : Bool;
      Especial_M236 : Bool;
      Bit_02_M236 : Bool;
      Retroceder_M236 : Bool;
      Retirar_M236 : Bool;
      Continuar_M236 : Bool;
      Entrar_M236 : Bool;
      EmiOK_M236 : Bool;
      FinLote_M237 : Bool;
      Especial_M237 : Bool;
      Bit_02_M237 : Bool;
      Retroceder_M237 : Bool;
      Retirar_M237 : Bool;
      Continuar_M237 : Bool;
      Entrar_M237 : Bool;
      EmiOK_M237 : Bool;
      FinLote_M238 : Bool;
      Especial_M238 : Bool;
      Bit_02_M238 : Bool;
      Retroceder_M238 : Bool;
      Retirar_M238 : Bool;
      Continuar_M238 : Bool;
      Entrar_M238 : Bool;
      EmiOK_M238 : Bool;
      FinLote_M239 : Bool;
      Especial_M239 : Bool;
      Bit_02_M239 : Bool;
      Retroceder_M239 : Bool;
      Retirar_M239 : Bool;
      Continuar_M239 : Bool;
      Entrar_M239 : Bool;
      EmiOK_M239 : Bool;
      FinLote_M240 : Bool;
      Especial_M240 : Bool;
      Bit_02_M240 : Bool;
      Retroceder_M240 : Bool;
      Retirar_M240 : Bool;
      Continuar_M240 : Bool;
      Entrar_M240 : Bool;
      EmiOK_M240 : Bool;
      FinLote_M241 : Bool;
      Especial_M241 : Bool;
      Bit_02_M241 : Bool;
      Retroceder_M241 : Bool;
      Retirar_M241 : Bool;
      Continuar_M241 : Bool;
      Entrar_M241 : Bool;
      EmiOK_M241 : Bool;
      FinLote_M242 : Bool;
      Especial_M242 : Bool;
      Bit_02_M242 : Bool;
      Retroceder_M242 : Bool;
      Retirar_M242 : Bool;
      Continuar_M242 : Bool;
      Entrar_M242 : Bool;
      EmiOK_M242 : Bool;
      FinLote_M243 : Bool;
      Especial_M243 : Bool;
      Bit_02_M243 : Bool;
      Retroceder_M243 : Bool;
      Retirar_M243 : Bool;
      Continuar_M243 : Bool;
      Entrar_M243 : Bool;
      EmiOK_M243 : Bool;
      FinLote_M244 : Bool;
      Especial_M244 : Bool;
      Bit_02_M244 : Bool;
      Retroceder_M244 : Bool;
      Retirar_M244 : Bool;
      Continuar_M244 : Bool;
      Entrar_M244 : Bool;
      EmiOK_M244 : Bool;
      FinLote_M245 : Bool;
      Especial_M245 : Bool;
      Bit_02_M245 : Bool;
      Retroceder_M245 : Bool;
      Retirar_M245 : Bool;
      Continuar_M245 : Bool;
      Entrar_M245 : Bool;
      EmiOK_M245 : Bool;
      FinLote_M246 : Bool;
      Especial_M246 : Bool;
      Bit_02_M246 : Bool;
      Retroceder_M246 : Bool;
      Retirar_M246 : Bool;
      Continuar_M246 : Bool;
      Entrar_M246 : Bool;
      EmiOK_M246 : Bool;
      FinLote_M247 : Bool;
      Especial_M247 : Bool;
      Bit_02_M247 : Bool;
      Retroceder_M247 : Bool;
      Retirar_M247 : Bool;
      Continuar_M247 : Bool;
      Entrar_M247 : Bool;
      EmiOK_M247 : Bool;
      FinLote_M248 : Bool;
      Especial_M248 : Bool;
      Bit_02_M248 : Bool;
      Retroceder_M248 : Bool;
      Retirar_M248 : Bool;
      Continuar_M248 : Bool;
      Entrar_M248 : Bool;
      EmiOK_M248 : Bool;
      FinLote_M249 : Bool;
      Especial_M249 : Bool;
      Bit_02_M249 : Bool;
      Retroceder_M249 : Bool;
      Retirar_M249 : Bool;
      Continuar_M249 : Bool;
      Entrar_M249 : Bool;
      EmiOK_M249 : Bool;
      FinLote_M250 : Bool;
      Especial_M250 : Bool;
      Bit_02_M250 : Bool;
      Retroceder_M250 : Bool;
      Retirar_M250 : Bool;
      Continuar_M250 : Bool;
      Entrar_M250 : Bool;
      EmiOK_M250 : Bool;
      FinLote_M251 : Bool;
      Especial_M251 : Bool;
      Bit_02_M251 : Bool;
      Retroceder_M251 : Bool;
      Retirar_M251 : Bool;
      Continuar_M251 : Bool;
      Entrar_M251 : Bool;
      EmiOK_M251 : Bool;
      FinLote_M252 : Bool;
      Especial_M252 : Bool;
      Bit_02_M252 : Bool;
      Retroceder_M252 : Bool;
      Retirar_M252 : Bool;
      Continuar_M252 : Bool;
      Entrar_M252 : Bool;
      EmiOK_M252 : Bool;
      FinLote_M253 : Bool;
      Especial_M253 : Bool;
      Bit_02_M253 : Bool;
      Retroceder_M253 : Bool;
      Retirar_M253 : Bool;
      Continuar_M253 : Bool;
      Entrar_M253 : Bool;
      EmiOK_M253 : Bool;
      FinLote_M254 : Bool;
      Especial_M254 : Bool;
      Bit_02_M254 : Bool;
      Retroceder_M254 : Bool;
      Retirar_M254 : Bool;
      Continuar_M254 : Bool;
      Entrar_M254 : Bool;
      EmiOK_M254 : Bool;
      FinLote_M255 : Bool;
      Especial_M255 : Bool;
      Bit_02_M255 : Bool;
      Retroceder_M255 : Bool;
      Retirar_M255 : Bool;
      Continuar_M255 : Bool;
      Entrar_M255 : Bool;
      EmiOK_M255 : Bool;
      FinLote_M256 : Bool;
      Especial_M256 : Bool;
      Bit_02_M256 : Bool;
      Retroceder_M256 : Bool;
      Retirar_M256 : Bool;
      Continuar_M256 : Bool;
      Entrar_M256 : Bool;
      EmiOK_M256 : Bool;
      FinLote_M257 : Bool;
      Especial_M257 : Bool;
      Bit_02_M257 : Bool;
      Retroceder_M257 : Bool;
      Retirar_M257 : Bool;
      Continuar_M257 : Bool;
      Entrar_M257 : Bool;
      EmiOK_M257 : Bool;
      FinLote_M258 : Bool;
      Especial_M258 : Bool;
      Bit_02_M258 : Bool;
      Retroceder_M258 : Bool;
      Retirar_M258 : Bool;
      Continuar_M258 : Bool;
      Entrar_M258 : Bool;
      EmiOK_M258 : Bool;
      FinLote_M259 : Bool;
      Especial_M259 : Bool;
      Bit_02_M259 : Bool;
      Retroceder_M259 : Bool;
      Retirar_M259 : Bool;
      Continuar_M259 : Bool;
      Entrar_M259 : Bool;
      EmiOK_M259 : Bool;
      FinLote_M260 : Bool;
      Especial_M260 : Bool;
      Bit_02_M260 : Bool;
      Retroceder_M260 : Bool;
      Retirar_M260 : Bool;
      Continuar_M260 : Bool;
      Entrar_M260 : Bool;
      EmiOK_M260 : Bool;
      FinLote_M261 : Bool;
      Especial_M261 : Bool;
      Bit_02_M261 : Bool;
      Retroceder_M261 : Bool;
      Retirar_M261 : Bool;
      Continuar_M261 : Bool;
      Entrar_M261 : Bool;
      EmiOK_M261 : Bool;
      FinLote_M262 : Bool;
      Especial_M262 : Bool;
      Bit_02_M262 : Bool;
      Retroceder_M262 : Bool;
      Retirar_M262 : Bool;
      Continuar_M262 : Bool;
      Entrar_M262 : Bool;
      EmiOK_M262 : Bool;
      FinLote_M263 : Bool;
      Especial_M263 : Bool;
      Bit_02_M263 : Bool;
      Retroceder_M263 : Bool;
      Retirar_M263 : Bool;
      Continuar_M263 : Bool;
      Entrar_M263 : Bool;
      EmiOK_M263 : Bool;
      FinLote_M264 : Bool;
      Especial_M264 : Bool;
      Bit_02_M264 : Bool;
      Retroceder_M264 : Bool;
      Retirar_M264 : Bool;
      Continuar_M264 : Bool;
      Entrar_M264 : Bool;
      EmiOK_M264 : Bool;
      FinLote_M265 : Bool;
      Especial_M265 : Bool;
      Bit_02_M265 : Bool;
      Retroceder_M265 : Bool;
      Retirar_M265 : Bool;
      Continuar_M265 : Bool;
      Entrar_M265 : Bool;
      EmiOK_M265 : Bool;
      FinLote_M266 : Bool;
      Especial_M266 : Bool;
      Bit_02_M266 : Bool;
      Retroceder_M266 : Bool;
      Retirar_M266 : Bool;
      Continuar_M266 : Bool;
      Entrar_M266 : Bool;
      EmiOK_M266 : Bool;
      FinLote_M267 : Bool;
      Especial_M267 : Bool;
      Bit_02_M267 : Bool;
      Retroceder_M267 : Bool;
      Retirar_M267 : Bool;
      Continuar_M267 : Bool;
      Entrar_M267 : Bool;
      EmiOK_M267 : Bool;
      FinLote_M268 : Bool;
      Especial_M268 : Bool;
      Bit_02_M268 : Bool;
      Retroceder_M268 : Bool;
      Retirar_M268 : Bool;
      Continuar_M268 : Bool;
      Entrar_M268 : Bool;
      EmiOK_M268 : Bool;
      FinLote_M269 : Bool;
      Especial_M269 : Bool;
      Bit_02_M269 : Bool;
      Retroceder_M269 : Bool;
      Retirar_M269 : Bool;
      Continuar_M269 : Bool;
      Entrar_M269 : Bool;
      EmiOK_M269 : Bool;
      FinLote_M270 : Bool;
      Especial_M270 : Bool;
      Bit_02_M270 : Bool;
      Retroceder_M270 : Bool;
      Retirar_M270 : Bool;
      Continuar_M270 : Bool;
      Entrar_M270 : Bool;
      EmiOK_M270 : Bool;
      FinLote_M271 : Bool;
      Especial_M271 : Bool;
      Bit_02_M271 : Bool;
      Retroceder_M271 : Bool;
      Retirar_M271 : Bool;
      Continuar_M271 : Bool;
      Entrar_M271 : Bool;
      EmiOK_M271 : Bool;
      FinLote_M272 : Bool;
      Especial_M272 : Bool;
      Bit_02_M272 : Bool;
      Retroceder_M272 : Bool;
      Retirar_M272 : Bool;
      Continuar_M272 : Bool;
      Entrar_M272 : Bool;
      EmiOK_M272 : Bool;
      FinLote_M273 : Bool;
      Especial_M273 : Bool;
      Bit_02_M273 : Bool;
      Retroceder_M273 : Bool;
      Retirar_M273 : Bool;
      Continuar_M273 : Bool;
      Entrar_M273 : Bool;
      EmiOK_M273 : Bool;
      FinLote_M274 : Bool;
      Especial_M274 : Bool;
      Bit_02_M274 : Bool;
      Retroceder_M274 : Bool;
      Retirar_M274 : Bool;
      Continuar_M274 : Bool;
      Entrar_M274 : Bool;
      EmiOK_M274 : Bool;
      FinLote_M275 : Bool;
      Especial_M275 : Bool;
      Bit_02_M275 : Bool;
      Retroceder_M275 : Bool;
      Retirar_M275 : Bool;
      Continuar_M275 : Bool;
      Entrar_M275 : Bool;
      EmiOK_M275 : Bool;
      FinLote_M276 : Bool;
      Especial_M276 : Bool;
      Bit_02_M276 : Bool;
      Retroceder_M276 : Bool;
      Retirar_M276 : Bool;
      Continuar_M276 : Bool;
      Entrar_M276 : Bool;
      EmiOK_M276 : Bool;
      FinLote_M277 : Bool;
      Especial_M277 : Bool;
      Bit_02_M277 : Bool;
      Retroceder_M277 : Bool;
      Retirar_M277 : Bool;
      Continuar_M277 : Bool;
      Entrar_M277 : Bool;
      EmiOK_M277 : Bool;
      FinLote_M278 : Bool;
      Especial_M278 : Bool;
      Bit_02_M278 : Bool;
      Retroceder_M278 : Bool;
      Retirar_M278 : Bool;
      Continuar_M278 : Bool;
      Entrar_M278 : Bool;
      EmiOK_M278 : Bool;
      FinLote_M279 : Bool;
      Especial_M279 : Bool;
      Bit_02_M279 : Bool;
      Retroceder_M279 : Bool;
      Retirar_M279 : Bool;
      Continuar_M279 : Bool;
      Entrar_M279 : Bool;
      EmiOK_M279 : Bool;
      FinLote_M280 : Bool;
      Especial_M280 : Bool;
      Bit_02_M280 : Bool;
      Retroceder_M280 : Bool;
      Retirar_M280 : Bool;
      Continuar_M280 : Bool;
      Entrar_M280 : Bool;
      EmiOK_M280 : Bool;
      FinLote_M281 : Bool;
      Especial_M281 : Bool;
      Bit_02_M281 : Bool;
      Retroceder_M281 : Bool;
      Retirar_M281 : Bool;
      Continuar_M281 : Bool;
      Entrar_M281 : Bool;
      EmiOK_M281 : Bool;
      FinLote_M282 : Bool;
      Especial_M282 : Bool;
      Bit_02_M282 : Bool;
      Retroceder_M282 : Bool;
      Retirar_M282 : Bool;
      Continuar_M282 : Bool;
      Entrar_M282 : Bool;
      EmiOK_M282 : Bool;
      FinLote_M283 : Bool;
      Especial_M283 : Bool;
      Bit_02_M283 : Bool;
      Retroceder_M283 : Bool;
      Retirar_M283 : Bool;
      Continuar_M283 : Bool;
      Entrar_M283 : Bool;
      EmiOK_M283 : Bool;
      FinLote_M284 : Bool;
      Especial_M284 : Bool;
      Bit_02_M284 : Bool;
      Retroceder_M284 : Bool;
      Retirar_M284 : Bool;
      Continuar_M284 : Bool;
      Entrar_M284 : Bool;
      EmiOK_M284 : Bool;
      FinLote_M285 : Bool;
      Especial_M285 : Bool;
      Bit_02_M285 : Bool;
      Retroceder_M285 : Bool;
      Retirar_M285 : Bool;
      Continuar_M285 : Bool;
      Entrar_M285 : Bool;
      EmiOK_M285 : Bool;
      FinLote_M286 : Bool;
      Especial_M286 : Bool;
      Bit_02_M286 : Bool;
      Retroceder_M286 : Bool;
      Retirar_M286 : Bool;
      Continuar_M286 : Bool;
      Entrar_M286 : Bool;
      EmiOK_M286 : Bool;
      FinLote_M287 : Bool;
      Especial_M287 : Bool;
      Bit_02_M287 : Bool;
      Retroceder_M287 : Bool;
      Retirar_M287 : Bool;
      Continuar_M287 : Bool;
      Entrar_M287 : Bool;
      EmiOK_M287 : Bool;
      FinLote_M288 : Bool;
      Especial_M288 : Bool;
      Bit_02_M288 : Bool;
      Retroceder_M288 : Bool;
      Retirar_M288 : Bool;
      Continuar_M288 : Bool;
      Entrar_M288 : Bool;
      EmiOK_M288 : Bool;
      FinLote_M289 : Bool;
      Especial_M289 : Bool;
      Bit_02_M289 : Bool;
      Retroceder_M289 : Bool;
      Retirar_M289 : Bool;
      Continuar_M289 : Bool;
      Entrar_M289 : Bool;
      EmiOK_M289 : Bool;
      FinLote_M290 : Bool;
      Especial_M290 : Bool;
      Bit_02_M290 : Bool;
      Retroceder_M290 : Bool;
      Retirar_M290 : Bool;
      Continuar_M290 : Bool;
      Entrar_M290 : Bool;
      EmiOK_M290 : Bool;
      FinLote_M291 : Bool;
      Especial_M291 : Bool;
      Bit_02_M291 : Bool;
      Retroceder_M291 : Bool;
      Retirar_M291 : Bool;
      Continuar_M291 : Bool;
      Entrar_M291 : Bool;
      EmiOK_M291 : Bool;
      FinLote_M292 : Bool;
      Especial_M292 : Bool;
      Bit_02_M292 : Bool;
      Retroceder_M292 : Bool;
      Retirar_M292 : Bool;
      Continuar_M292 : Bool;
      Entrar_M292 : Bool;
      EmiOK_M292 : Bool;
      FinLote_M293 : Bool;
      Especial_M293 : Bool;
      Bit_02_M293 : Bool;
      Retroceder_M293 : Bool;
      Retirar_M293 : Bool;
      Continuar_M293 : Bool;
      Entrar_M293 : Bool;
      EmiOK_M293 : Bool;
      FinLote_M294 : Bool;
      Especial_M294 : Bool;
      Bit_02_M294 : Bool;
      Retroceder_M294 : Bool;
      Retirar_M294 : Bool;
      Continuar_M294 : Bool;
      Entrar_M294 : Bool;
      EmiOK_M294 : Bool;
      FinLote_M295 : Bool;
      Especial_M295 : Bool;
      Bit_02_M295 : Bool;
      Retroceder_M295 : Bool;
      Retirar_M295 : Bool;
      Continuar_M295 : Bool;
      Entrar_M295 : Bool;
      EmiOK_M295 : Bool;
      FinLote_M296 : Bool;
      Especial_M296 : Bool;
      Bit_02_M296 : Bool;
      Retroceder_M296 : Bool;
      Retirar_M296 : Bool;
      Continuar_M296 : Bool;
      Entrar_M296 : Bool;
      EmiOK_M296 : Bool;
      FinLote_M297 : Bool;
      Especial_M297 : Bool;
      Bit_02_M297 : Bool;
      Retroceder_M297 : Bool;
      Retirar_M297 : Bool;
      Continuar_M297 : Bool;
      Entrar_M297 : Bool;
      EmiOK_M297 : Bool;
      FinLote_M298 : Bool;
      Especial_M298 : Bool;
      Bit_02_M298 : Bool;
      Retroceder_M298 : Bool;
      Retirar_M298 : Bool;
      Continuar_M298 : Bool;
      Entrar_M298 : Bool;
      EmiOK_M298 : Bool;
      FinLote_M299 : Bool;
      Especial_M299 : Bool;
      Bit_02_M299 : Bool;
      Retroceder_M299 : Bool;
      Retirar_M299 : Bool;
      Continuar_M299 : Bool;
      Entrar_M299 : Bool;
      EmiOK_M299 : Bool;
      FinLote_M300 : Bool;
      Especial_M300 : Bool;
      Bit_02_M300 : Bool;
      Retroceder_M300 : Bool;
      Retirar_M300 : Bool;
      Continuar_M300 : Bool;
      Entrar_M300 : Bool;
      EmiOK_M300 : Bool;
      FinLote_M301 : Bool;
      Especial_M301 : Bool;
      Bit_02_M301 : Bool;
      Retroceder_M301 : Bool;
      Retirar_M301 : Bool;
      Continuar_M301 : Bool;
      Entrar_M301 : Bool;
      EmiOK_M301 : Bool;
      FinLote_M302 : Bool;
      Especial_M302 : Bool;
      Bit_02_M302 : Bool;
      Retroceder_M302 : Bool;
      Retirar_M302 : Bool;
      Continuar_M302 : Bool;
      Entrar_M302 : Bool;
      EmiOK_M302 : Bool;
      FinLote_M303 : Bool;
      Especial_M303 : Bool;
      Bit_02_M303 : Bool;
      Retroceder_M303 : Bool;
      Retirar_M303 : Bool;
      Continuar_M303 : Bool;
      Entrar_M303 : Bool;
      EmiOK_M303 : Bool;
      FinLote_M304 : Bool;
      Especial_M304 : Bool;
      Bit_02_M304 : Bool;
      Retroceder_M304 : Bool;
      Retirar_M304 : Bool;
      Continuar_M304 : Bool;
      Entrar_M304 : Bool;
      EmiOK_M304 : Bool;
      FinLote_M305 : Bool;
      Especial_M305 : Bool;
      Bit_02_M305 : Bool;
      Retroceder_M305 : Bool;
      Retirar_M305 : Bool;
      Continuar_M305 : Bool;
      Entrar_M305 : Bool;
      EmiOK_M305 : Bool;
      FinLote_M306 : Bool;
      Especial_M306 : Bool;
      Bit_02_M306 : Bool;
      Retroceder_M306 : Bool;
      Retirar_M306 : Bool;
      Continuar_M306 : Bool;
      Entrar_M306 : Bool;
      EmiOK_M306 : Bool;
      FinLote_M307 : Bool;
      Especial_M307 : Bool;
      Bit_02_M307 : Bool;
      Retroceder_M307 : Bool;
      Retirar_M307 : Bool;
      Continuar_M307 : Bool;
      Entrar_M307 : Bool;
      EmiOK_M307 : Bool;
      FinLote_M308 : Bool;
      Especial_M308 : Bool;
      Bit_02_M308 : Bool;
      Retroceder_M308 : Bool;
      Retirar_M308 : Bool;
      Continuar_M308 : Bool;
      Entrar_M308 : Bool;
      EmiOK_M308 : Bool;
      FinLote_M309 : Bool;
      Especial_M309 : Bool;
      Bit_02_M309 : Bool;
      Retroceder_M309 : Bool;
      Retirar_M309 : Bool;
      Continuar_M309 : Bool;
      Entrar_M309 : Bool;
      EmiOK_M309 : Bool;
      FinLote_M310 : Bool;
      Especial_M310 : Bool;
      Bit_02_M310 : Bool;
      Retroceder_M310 : Bool;
      Retirar_M310 : Bool;
      Continuar_M310 : Bool;
      Entrar_M310 : Bool;
      EmiOK_M310 : Bool;
      FinLote_M311 : Bool;
      Especial_M311 : Bool;
      Bit_02_M311 : Bool;
      Retroceder_M311 : Bool;
      Retirar_M311 : Bool;
      Continuar_M311 : Bool;
      Entrar_M311 : Bool;
      EmiOK_M311 : Bool;
      FinLote_M312 : Bool;
      Especial_M312 : Bool;
      Bit_02_M312 : Bool;
      Retroceder_M312 : Bool;
      Retirar_M312 : Bool;
      Continuar_M312 : Bool;
      Entrar_M312 : Bool;
      EmiOK_M312 : Bool;
      FinLote_M313 : Bool;
      Especial_M313 : Bool;
      Bit_02_M313 : Bool;
      Retroceder_M313 : Bool;
      Retirar_M313 : Bool;
      Continuar_M313 : Bool;
      Entrar_M313 : Bool;
      EmiOK_M313 : Bool;
      FinLote_M314 : Bool;
      Especial_M314 : Bool;
      Bit_02_M314 : Bool;
      Retroceder_M314 : Bool;
      Retirar_M314 : Bool;
      Continuar_M314 : Bool;
      Entrar_M314 : Bool;
      EmiOK_M314 : Bool;
      FinLote_M315 : Bool;
      Especial_M315 : Bool;
      Bit_02_M315 : Bool;
      Retroceder_M315 : Bool;
      Retirar_M315 : Bool;
      Continuar_M315 : Bool;
      Entrar_M315 : Bool;
      EmiOK_M315 : Bool;
      FinLote_M316 : Bool;
      Especial_M316 : Bool;
      Bit_02_M316 : Bool;
      Retroceder_M316 : Bool;
      Retirar_M316 : Bool;
      Continuar_M316 : Bool;
      Entrar_M316 : Bool;
      EmiOK_M316 : Bool;
      FinLote_M317 : Bool;
      Especial_M317 : Bool;
      Bit_02_M317 : Bool;
      Retroceder_M317 : Bool;
      Retirar_M317 : Bool;
      Continuar_M317 : Bool;
      Entrar_M317 : Bool;
      EmiOK_M317 : Bool;
      FinLote_M318 : Bool;
      Especial_M318 : Bool;
      Bit_02_M318 : Bool;
      Retroceder_M318 : Bool;
      Retirar_M318 : Bool;
      Continuar_M318 : Bool;
      Entrar_M318 : Bool;
      EmiOK_M318 : Bool;
      FinLote_M319 : Bool;
      Especial_M319 : Bool;
      Bit_02_M319 : Bool;
      Retroceder_M319 : Bool;
      Retirar_M319 : Bool;
      Continuar_M319 : Bool;
      Entrar_M319 : Bool;
      EmiOK_M319 : Bool;
      FinLote_M320 : Bool;
      Especial_M320 : Bool;
      Bit_02_M320 : Bool;
      Retroceder_M320 : Bool;
      Retirar_M320 : Bool;
      Continuar_M320 : Bool;
      Entrar_M320 : Bool;
      EmiOK_M320 : Bool;
      FinLote_M321 : Bool;
      Especial_M321 : Bool;
      Bit_02_M321 : Bool;
      Retroceder_M321 : Bool;
      Retirar_M321 : Bool;
      Continuar_M321 : Bool;
      Entrar_M321 : Bool;
      EmiOK_M321 : Bool;
      FinLote_M322 : Bool;
      Especial_M322 : Bool;
      Bit_02_M322 : Bool;
      Retroceder_M322 : Bool;
      Retirar_M322 : Bool;
      Continuar_M322 : Bool;
      Entrar_M322 : Bool;
      EmiOK_M322 : Bool;
      FinLote_M323 : Bool;
      Especial_M323 : Bool;
      Bit_02_M323 : Bool;
      Retroceder_M323 : Bool;
      Retirar_M323 : Bool;
      Continuar_M323 : Bool;
      Entrar_M323 : Bool;
      EmiOK_M323 : Bool;
      FinLote_M324 : Bool;
      Especial_M324 : Bool;
      Bit_02_M324 : Bool;
      Retroceder_M324 : Bool;
      Retirar_M324 : Bool;
      Continuar_M324 : Bool;
      Entrar_M324 : Bool;
      EmiOK_M324 : Bool;
      FinLote_M325 : Bool;
      Especial_M325 : Bool;
      Bit_02_M325 : Bool;
      Retroceder_M325 : Bool;
      Retirar_M325 : Bool;
      Continuar_M325 : Bool;
      Entrar_M325 : Bool;
      EmiOK_M325 : Bool;
      FinLote_M326 : Bool;
      Especial_M326 : Bool;
      Bit_02_M326 : Bool;
      Retroceder_M326 : Bool;
      Retirar_M326 : Bool;
      Continuar_M326 : Bool;
      Entrar_M326 : Bool;
      EmiOK_M326 : Bool;
      FinLote_M327 : Bool;
      Especial_M327 : Bool;
      Bit_02_M327 : Bool;
      Retroceder_M327 : Bool;
      Retirar_M327 : Bool;
      Continuar_M327 : Bool;
      Entrar_M327 : Bool;
      EmiOK_M327 : Bool;
      FinLote_M328 : Bool;
      Especial_M328 : Bool;
      Bit_02_M328 : Bool;
      Retroceder_M328 : Bool;
      Retirar_M328 : Bool;
      Continuar_M328 : Bool;
      Entrar_M328 : Bool;
      EmiOK_M328 : Bool;
      FinLote_M329 : Bool;
      Especial_M329 : Bool;
      Bit_02_M329 : Bool;
      Retroceder_M329 : Bool;
      Retirar_M329 : Bool;
      Continuar_M329 : Bool;
      Entrar_M329 : Bool;
      EmiOK_M329 : Bool;
      FinLote_M330 : Bool;
      Especial_M330 : Bool;
      Bit_02_M330 : Bool;
      Retroceder_M330 : Bool;
      Retirar_M330 : Bool;
      Continuar_M330 : Bool;
      Entrar_M330 : Bool;
      EmiOK_M330 : Bool;
      FinLote_M331 : Bool;
      Especial_M331 : Bool;
      Bit_02_M331 : Bool;
      Retroceder_M331 : Bool;
      Retirar_M331 : Bool;
      Continuar_M331 : Bool;
      Entrar_M331 : Bool;
      EmiOK_M331 : Bool;
      FinLote_M332 : Bool;
      Especial_M332 : Bool;
      Bit_02_M332 : Bool;
      Retroceder_M332 : Bool;
      Retirar_M332 : Bool;
      Continuar_M332 : Bool;
      Entrar_M332 : Bool;
      EmiOK_M332 : Bool;
      FinLote_M333 : Bool;
      Especial_M333 : Bool;
      Bit_02_M333 : Bool;
      Retroceder_M333 : Bool;
      Retirar_M333 : Bool;
      Continuar_M333 : Bool;
      Entrar_M333 : Bool;
      EmiOK_M333 : Bool;
      FinLote_M334 : Bool;
      Especial_M334 : Bool;
      Bit_02_M334 : Bool;
      Retroceder_M334 : Bool;
      Retirar_M334 : Bool;
      Continuar_M334 : Bool;
      Entrar_M334 : Bool;
      EmiOK_M334 : Bool;
      FinLote_M335 : Bool;
      Especial_M335 : Bool;
      Bit_02_M335 : Bool;
      Retroceder_M335 : Bool;
      Retirar_M335 : Bool;
      Continuar_M335 : Bool;
      Entrar_M335 : Bool;
      EmiOK_M335 : Bool;
      FinLote_M336 : Bool;
      Especial_M336 : Bool;
      Bit_02_M336 : Bool;
      Retroceder_M336 : Bool;
      Retirar_M336 : Bool;
      Continuar_M336 : Bool;
      Entrar_M336 : Bool;
      EmiOK_M336 : Bool;
      FinLote_M337 : Bool;
      Especial_M337 : Bool;
      Bit_02_M337 : Bool;
      Retroceder_M337 : Bool;
      Retirar_M337 : Bool;
      Continuar_M337 : Bool;
      Entrar_M337 : Bool;
      EmiOK_M337 : Bool;
      FinLote_M338 : Bool;
      Especial_M338 : Bool;
      Bit_02_M338 : Bool;
      Retroceder_M338 : Bool;
      Retirar_M338 : Bool;
      Continuar_M338 : Bool;
      Entrar_M338 : Bool;
      EmiOK_M338 : Bool;
      FinLote_M339 : Bool;
      Especial_M339 : Bool;
      Bit_02_M339 : Bool;
      Retroceder_M339 : Bool;
      Retirar_M339 : Bool;
      Continuar_M339 : Bool;
      Entrar_M339 : Bool;
      EmiOK_M339 : Bool;
      FinLote_M340 : Bool;
      Especial_M340 : Bool;
      Bit_02_M340 : Bool;
      Retroceder_M340 : Bool;
      Retirar_M340 : Bool;
      Continuar_M340 : Bool;
      Entrar_M340 : Bool;
      EmiOK_M340 : Bool;
      FinLote_M341 : Bool;
      Especial_M341 : Bool;
      Bit_02_M341 : Bool;
      Retroceder_M341 : Bool;
      Retirar_M341 : Bool;
      Continuar_M341 : Bool;
      Entrar_M341 : Bool;
      EmiOK_M341 : Bool;
      FinLote_M342 : Bool;
      Especial_M342 : Bool;
      Bit_02_M342 : Bool;
      Retroceder_M342 : Bool;
      Retirar_M342 : Bool;
      Continuar_M342 : Bool;
      Entrar_M342 : Bool;
      EmiOK_M342 : Bool;
      FinLote_M343 : Bool;
      Especial_M343 : Bool;
      Bit_02_M343 : Bool;
      Retroceder_M343 : Bool;
      Retirar_M343 : Bool;
      Continuar_M343 : Bool;
      Entrar_M343 : Bool;
      EmiOK_M343 : Bool;
      FinLote_M344 : Bool;
      Especial_M344 : Bool;
      Bit_02_M344 : Bool;
      Retroceder_M344 : Bool;
      Retirar_M344 : Bool;
      Continuar_M344 : Bool;
      Entrar_M344 : Bool;
      EmiOK_M344 : Bool;
      FinLote_M345 : Bool;
      Especial_M345 : Bool;
      Bit_02_M345 : Bool;
      Retroceder_M345 : Bool;
      Retirar_M345 : Bool;
      Continuar_M345 : Bool;
      Entrar_M345 : Bool;
      EmiOK_M345 : Bool;
      FinLote_M346 : Bool;
      Especial_M346 : Bool;
      Bit_02_M346 : Bool;
      Retroceder_M346 : Bool;
      Retirar_M346 : Bool;
      Continuar_M346 : Bool;
      Entrar_M346 : Bool;
      EmiOK_M346 : Bool;
      FinLote_M347 : Bool;
      Especial_M347 : Bool;
      Bit_02_M347 : Bool;
      Retroceder_M347 : Bool;
      Retirar_M347 : Bool;
      Continuar_M347 : Bool;
      Entrar_M347 : Bool;
      EmiOK_M347 : Bool;
      FinLote_M348 : Bool;
      Especial_M348 : Bool;
      Bit_02_M348 : Bool;
      Retroceder_M348 : Bool;
      Retirar_M348 : Bool;
      Continuar_M348 : Bool;
      Entrar_M348 : Bool;
      EmiOK_M348 : Bool;
      FinLote_M349 : Bool;
      Especial_M349 : Bool;
      Bit_02_M349 : Bool;
      Retroceder_M349 : Bool;
      Retirar_M349 : Bool;
      Continuar_M349 : Bool;
      Entrar_M349 : Bool;
      EmiOK_M349 : Bool;
      FinLote_M350 : Bool;
      Especial_M350 : Bool;
      Bit_02_M350 : Bool;
      Retroceder_M350 : Bool;
      Retirar_M350 : Bool;
      Continuar_M350 : Bool;
      Entrar_M350 : Bool;
      EmiOK_M350 : Bool;
      FinLote_M351 : Bool;
      Especial_M351 : Bool;
      Bit_02_M351 : Bool;
      Retroceder_M351 : Bool;
      Retirar_M351 : Bool;
      Continuar_M351 : Bool;
      Entrar_M351 : Bool;
      EmiOK_M351 : Bool;
      FinLote_M352 : Bool;
      Especial_M352 : Bool;
      Bit_02_M352 : Bool;
      Retroceder_M352 : Bool;
      Retirar_M352 : Bool;
      Continuar_M352 : Bool;
      Entrar_M352 : Bool;
      EmiOK_M352 : Bool;
      FinLote_M353 : Bool;
      Especial_M353 : Bool;
      Bit_02_M353 : Bool;
      Retroceder_M353 : Bool;
      Retirar_M353 : Bool;
